// =============================================================================
// 段 2: 三轴伺服电流监测（仅使能时读 AD，%IW×%ID/1e6）
// %IW10/%ID4=俯仰, %IW20/%ID9=方位, %IW30/%ID14=倾斜
// =============================================================================
IF Axis1Status.bServo_Enable THEN
	rELCurrent:=DINT_TO_REAL((INT_TO_DINT(%IW10)* %ID4))/1000000.0;  //俯仰轴电流监测
ELSE
	rELCurrent:=0;
END_IF

IF Axis2Status.bServo_Enable THEN
	rAzCurrent:=DINT_TO_REAL((INT_TO_DINT(%IW20)* %ID9))/1000000.0;  //方位轴电流监测
ELSE
	rAzCurrent:=0;
END_IF

IF Axis3Status.bServo_Enable THEN
	rTlCurrent:=DINT_TO_REAL((INT_TO_DINT(%IW30)* %ID14))/1000000.0;  //倾斜轴电流监测
ELSE
	rTlCurrent:=0;
END_IF

// =============================================================================
// 段 3: 跟踪误差（供 SpiralScan 判断扫描方向与完成度）
// mode2 指向: 命令位置 vs 实际位置
// mode4 程引: 插值目标+偏置 vs 实际位置（含手动/自跟踪偏置）
// =============================================================================
IF Axis2Remote.iMode = 2 THEN
	AzError:=(-1) * (Axis2Remote.rPosCmd-rFctPosReal_2);
	ElError:=Axis1Remote.rPosCmd-rFctPosReal_1;	
END_IF

IF Axis2Remote.iMode = 4 THEN
	AzError:=rFctPosReal_2-RealTimePosCal.rInterazPos-(az_ctrl_1.rStepBias+az_ctrl_1.rAuToStepBias);
	ElError:=RealTimePosCal.rInterElPos-rFctPosReal_1+ (El_ctrl_1.rStepBias+EL_ctrl_1.rAuToStepBias);
END_IF
(*
rAzErrorReal := rAzErrorReal + rAlpha * (AzError - rAzErrorReal);
rElErrorReal := rElErrorReal + rAlpha * (ElError - rElErrorReal);
*)

// =============================================================================
// 段 4: 远控故障复位（Modbus bCommReset → GVL.bError_Reset）
// =============================================================================
IF NOT GVL.bLocalCtrl THEN
	IF Modbus_Slave.bCommReset THEN
		GVL.bError_Reset:=TRUE;
	ELSE
		GVL.bError_Reset:=FALSE;
	END_IF
END_IF

// =============================================================================
// 段 5: 远控 rPosCmd 赋值（含 AGC 搜索偏置或测试扫描偏置）
// 非 bSearch: Modbus 目标 + eltest/aztest
// bSearch:   Modbus 目标 + *_ctrl_1 的 rSearchNextStepTarget_tb
// =============================================================================
IF NOT modbus_slave.bSearch THEN
	Axis1Remote.rPosCmd:=Modbus_Slave.rPosCmd_1 + eltest;
	Axis2Remote.rPosCmd:=Modbus_Slave.rPosCmd_2 - aztest;
ELSE
	Axis1Remote.rPosCmd:=Modbus_Slave.rPosCmd_1 + El_ctrl_1.rSearchNextStepTarget_tb;
	Axis2Remote.rPosCmd:=Modbus_Slave.rPosCmd_2 + Az_ctrl_1.rSearchNextStepTarget_tb;
END_IF

// =============================================================================
// 段 6: 远控三轴命令参量 — Modbus_Slave → AxisXRemote（核心汇总）
// 俯仰/方位 rPosCmd 已在段 5 赋值；此处写 mode/速度/PID/加减速等
// =============================================================================
Axis1Remote.iMode:=Modbus_Slave.iMode_1;
Axis1Remote.rVelCmd:=Modbus_Slave.rVelcmd_1;
//Axis1Remote.rPosCmd:=Modbus_Slave.rPosCmd_1;
Axis1Remote.rP:=Modbus_Slave.rP_1;
Axis1Remote.rI:=Modbus_Slave.rI_1;
Axis1Remote.rD:=Modbus_Slave.rD_1;
Axis1Remote.rPIDThre:=Modbus_Slave.rThreshold_1;
Axis1Remote.rAcceleration:=Modbus_Slave.rAcceleration_1;
Axis1Remote.rDeceleration:=Modbus_Slave.rDeceleration_1;
Axis1Remote.rVel_Limit:=Modbus_Slave.rVelLim_1;

Axis2Remote.iMode:=Modbus_Slave.iMode_2;
Axis2Remote.rVelCmd:=Modbus_Slave.rVelcmd_2;
//Axis2Remote.rPosCmd:=Modbus_Slave.rPosCmd_2;
Axis2Remote.rP:=Modbus_Slave.rP_2;
Axis2Remote.rI:=Modbus_Slave.rI_2;
Axis2Remote.rD:=Modbus_Slave.rD_2;
Axis2Remote.rPIDThre:=Modbus_Slave.rThreshold_2;
Axis2Remote.rAcceleration:=Modbus_Slave.rAcceleration_2;
Axis2Remote.rDeceleration:=Modbus_Slave.rDeceleration_2;
Axis2Remote.rVel_Limit:=Modbus_Slave.rVelLim_2;

Axis3Remote.iMode:=Modbus_Slave.iMode_3;
Axis3Remote.rVelCmd:=Modbus_Slave.rVelcmd_3;
Axis3Remote.rPosCmd:=Modbus_Slave.rPosCmd_3;
Axis3Remote.rP:=Modbus_Slave.rP_3;
Axis3Remote.rI:=Modbus_Slave.rI_3;
Axis3Remote.rD:=Modbus_Slave.rD_3;
Axis3Remote.rPIDThre:=Modbus_Slave.rThreshold_3;
Axis3Remote.rAcceleration:=Modbus_Slave.rAcceleration_3;
Axis3Remote.rDeceleration:=Modbus_Slave.rDeceleration_3;

(* 本控 HMI 赋值块已注释，本控参数由其他 POU 写入 AxisXLocal *)

// =============================================================================
// 段 7: 俯仰预限位 → Error_code 201(正)/202(负)，置位上报标志
// bPrelimit_1 由硬件 IO 映射；触发后根据当前位置方向区分正负限位
// =============================================================================
IF bPrelimit_1 THEN
	IF rFctPosReal_1>0 THEN
		bPrelimit_Positive_1:=TRUE;
		Error_code:=201;
	ELSE
		bPrelimit_Negative_1:=TRUE;
		Error_code:=202;
	END_IF;
ELSE
	bPrelimit_Negative_1:=FALSE;
	bPrelimit_Positive_1:=FALSE;
	;
END_IF

// =============================================================================
// 段 8: 方位预限位（仅置标志，Error_code 203/204 已注释）
// =============================================================================
IF bPrelimit_2 THEN
	IF rFctPosReal_2>0 THEN
		//Error_code:=203;
		bPrelimit_Positive_2:=TRUE;;
	ELSE
		//Error_code:=204;
		bPrelimit_Negative_2:=TRUE;;
	END_IF;
ELSE
	bPrelimit_Negative_2:=FALSE;
	bPrelimit_Positive_2:=FALSE;
	;
END_IF

// =============================================================================
// 段 9: 扫描找到中心 — 基带锁 且 Eb/N0>rEbN0LockThre 且 √(Ua²+Ue²)<=rErrorThre
// =============================================================================
bBaseLock := (READ_485.recBuf[1] = 1);
bErrorLock  := (SQRT(GVL.Chan1Ua * GVL.Chan1Ua + GVL.Chan1Ue * GVL.Chan1Ue) <= PersistentVars.rErrorThre);
bLockSearch := (READ_485.Chan1EB_N0 > PersistentVars.rEbN0LockThre) AND bBaseLock AND bErrorLock;

// =============================================================================
// 段 10: 启扫 — 双轴程引、未自跟踪、基带锁连续 2s（200×10ms）触发一次
// 扫描过程中允许短暂掉锁；找到合格点后本程引周期内不再重扫
// 退出程引则清锁存
// =============================================================================
IF Axis1Remote.iMode = 4 AND Axis2Remote.iMode = 4 THEN
	IF NOT GVL.bStartTrack AND NOT bScanRun AND NOT bScanFound THEN
		IF bBaseLock THEN
			icountBaseLock := icountBaseLock + 1;
			IF icountBaseLock >= 200 THEN
				icountBaseLock := 200;
				bScanRun := TRUE;
			END_IF
		ELSE
			icountBaseLock := 0;
		END_IF
	ELSE
		icountBaseLock := 0;
	END_IF
	enable := bScanRun AND NOT GVL.bStartTrack;
ELSE
	enable := FALSE;
	bScanRun := FALSE;
	bScanDoneOnce := FALSE;
	bScanFound := FALSE;
	az_latch := 0.0;
	el_latch := 0.0;
	icountBaseLock := 0;
END_IF

// 螺旋局部参数（与直线 PersistentVars.rStep 量纲不同：此处为每格周期数）
IF rdelta < 1.0E-6 THEN
	rdelta := 0.25;
END_IF
IF rStep < 1.0E-6 THEN
	rStep := 12.0;
END_IF

// =============================================================================
// 段 11: 调用扫描 FB — 直线或螺旋；locked=找到中心，连续10拍（约100ms）锁存
// =============================================================================
IF NOT PersistentVars.bSearchType THEN
	fbScan(
		enable      := enable,
		delta       := PersistentVars.rAzScanRange,
		delta1      := PersistentVars.rElScanRange,
		n_steps     := PersistentVars.rStep,
		agc      := READ_485.Chan1EB_N0,
		locked     := bLockSearch,
		AzError := AzError,
		elError := elError,
		bTrackState := GVL.bStartTrack,
		azimuth     => az_out,
		elevation   => el_out,
		done        => done_out,
		bType  =>bType_out
	);
ELSE
	fbScan1(
		enable      := enable,
		delta       := rdelta,
		n_steps     := rStep,
		agc      := READ_485.Chan1EB_N0,
		locked     := bLockSearch,
		AzError := AzError,
		elError := elError,
		azimuth     => az_out,
		elevation   => el_out,
		done        => done_out,
		bType  =>bType_out
	);
END_IF

// 扫描结束：找到则锁存 -Error；未找到锁存 0。此后 az_out/el_out 用锁存值
IF bScanRun AND done_out THEN
	bScanRun := FALSE;
	bScanDoneOnce := TRUE;
	IF bType_out THEN
		az_latch := az_out;
		el_latch := el_out;
		bScanFound := TRUE;
	ELSE
		az_latch := 0.0;
		el_latch := 0.0;
		bScanFound := FALSE;
	END_IF
END_IF
IF GVL.bStartTrack AND bScanRun THEN
	bScanRun := FALSE;
	bScanDoneOnce := TRUE;
END_IF
IF NOT bScanRun THEN
	az_out := az_latch;
	el_out := el_latch;
END_IF

// =============================================================================
// 段 12: 自跟踪只跟 ACU HR[7].B10（上升沿开、下降沿关），扫描结束不置位
// =============================================================================
IF Axis1Remote.iMode = 4 AND Axis2Remote.iMode = 4 THEN
	RiseEdge(CLK := Modbus_Slave.bStartTrackAcu);
	FallEdge(CLK := Modbus_Slave.bStartTrackAcu);
	IF RiseEdge.Q THEN
		GVL.bStartTrack := TRUE;
	END_IF;
	IF FallEdge.Q THEN
		GVL.bStartTrack := FALSE;
	END_IF;
ELSE
	GVL.bStartTrack := Modbus_Slave.bStartTrackAcu;
	icountLostLocking := 0;
	icountLostLocking1 := 0;
	Iconutwait := 0;
END_IF

(* fbScantest 测试块已注释 *)

(* PHASE_CAL_HOOK: once per 10 ms, LAST call. *)
PRG_PhaseCalibration();
                  
END_PROGRAM

FUNCTION_BLOCK PID_1
VAR_INPUT
    rTarget : REAL;       (* 设定值 *)
    rFeedback : REAL;       (* 反馈值 *)
	rPosLimPositive:LREAL;//位置正限位
	rPosLimNegative:LREAL;//位置反限位
	rKp:REAL;     //比例增益
	rKi:REAL;     //积分增益
	rKd:REAL;     //微分增益
	iThreshold:INT;//积分项开启的位置阈值
	bPIDEnable:BOOL:=TRUE;//PID使能
	rVelLim:LREAL;//速度限制
END_VAR
VAR_OUTPUT
    rPIDOutput : LREAL:=0;         //带方向的输出速度

END_VAR
VAR
	//rPIDOutPut: REAL:=0.0;
	rLastError: LREAL:=0.0;(*上一次误差*)
	rErrorNow:LREAL:=0.0;(*当前误差*)
    rIntegralNew : LREAL := 0.0; (* 积分项 *)
    rDerivativeNew : LREAL := 0.0; (* 微分项 *)
	rDelta: LREAL;(*增量*)
	rProportionNew: LREAL;
	
	//iAzPIDEnable: INT;
END_VAR

                    
IF (bPIDEnable>0) THEN //如果PID使能
	IF rTarget=rFeedback THEN
		rPIDOutput:=0;	
	ELSE
	
		rErrorNow:=rTarget-rFeedback;//计算当前误差 en
		rProportionNew:=rErrorNow;//比例项
		//积分项
		IF rFeedback>rPosLimNegative AND rFeedback<rPosLimPositive THEN //若在软限位之内，工作时开启积分项
			IF (ABS(rTarget-rFeedback)<iThreshold OR iThreshold = -1) THEN//位置差小于积分阈值开始积分，或者设置阈值为-1，不启用这个控制
				rIntegralNew:= rIntegralNew+rErrorNow; //积分项
			ELSE
				rIntegralNew:=0;
			END_IF;
		ELSE //不在软限位范围内,则积分项为0
			rIntegralNew:=0;
		END_IF

		//PID输出
		rPIDOutPut:=rKp*rProportionNew+rKi*rIntegralNew;


		//PID限速
		
			IF rPIDOutput<(-rVelLim) THEN
				rPIDOutput:=-rVelLim;
			ELSIF rPIDOutput>rVelLim THEN
				rPIDOutput:=rVelLim;
			END_IF
		
		
		IF rFeedback>rPosLimPositive AND rPIDOutput>0 THEN 
			rPIDOutput:=0;
		END_IF
		IF rFeedback<rPosLimNegative AND rPIDOutput<0 THEN
			rPIDOutput:=0;
		END_IF
		
		rLastError:=rErrorNow;//将当前误差赋值给上一次误差
		
	END_IF
ELSE//非使能清零PID各项
	rProportionNew:=0.0;
	rIntegralNew:=0.0;
	rPIDOutput:=0.0;
END_IF










                  
END_FUNCTION_BLOCK

PROGRAM AutoTrackingCal
VAR
	rChanUa:REAL;//自跟踪采用的跟踪接收机ua
	rChanUe:REAL;//自跟踪采用的跟踪接收机ue
	rChanAGC:REAL;//自跟踪采用的跟踪接收机AGC
	bChanLock:BOOL;//频道是否锁定
	iCountATLock:INT;//自跟踪锁定
	iState:INT;//Case选择变量
	
	rAzSum:LREAL;//方位累计量
	rElSum:LREAL;//俯仰累积量
	
	rDirSenFac:REAL:=12;
	rCurentEl:LREAL;//当前俯仰角
	rk: LREAL:=1/15.0;
	
	rChanUaLocal:REAL;//自跟踪采用的跟踪接收机ua
	rChanUeLocal:REAL;//自跟踪采用的跟踪接收机ue
END_VAR

                    (*
IF iState=1 THEN
	rChanUa:=GVL.Chan1Ua;
	rChanUe:=GVL.Chan1Ue;
	rChanAGC:=GVL.Chan1AGC;
	bChanLock:=TRUE;
ELSIF iState=2 THEN
	rChanUa:=GVL.Chan2Ua;
	rChanUe:=GVL.Chan2Ue;
	rChanAGC:=GVL.Chan2AGC;
	bChanLock:=TRUE;
ELSE 
	bChanLock:=FALSE;
END_IF
*)

//iState:=modbusSlave.Trace_Num;//跟踪支路选择
iState:=1;

CASE iState OF 
	1://使用跟踪接收机1 且锁定标识为True
		//
		//bChanLock:=TRUE;
		//方位
		IF GVL.bStartTrack AND (GVL.Chan1Lock OR Securitycheck.bErrorLock) THEN
			//根据误差电压正负决定拉偏方向
			rChanUa:=GVL.Chan1Ua;
			//rChanUa:=rChanUa/UDINT_TO_REAL(modbusSlave.DirSenFac);
			rChanUa:=rChanUa/rDirSenFac;
			rCurentEl:=(rFctPosReal_1-90)*3.1415926535897/180.0;
			rChanUa:=rChanUa/COS(rCurentEl);
			
			//俯仰
			rChanUe:=GVL.Chan1Ue;
			//rChanUe:=rChanUe/UDINT_TO_REAL(modbusSlave.DirSenFac);;
			rChanUe:=rChanUe/rDirSenFac;
			rChanAGC:=GVL.Chan1AGC;
			
			//累积量
			rAzSum:=rAzSum+rk*rChanUa/1000.0;
			rElSum:=rElSum+rk*rChanUe/1000.0;
		ELSE
			rAzSum:=0;
			rElSum:=0;
			rChanUa:=0;
			rChanUe:=0;
		END_IF
		
	2://使用跟踪接收机2 且锁定标识为True
		//
		//bChanLock:=TRUE;
		rChanUa:=GVL.Chan2Ua;
		rChanUe:=GVL.Chan2Ue;
		rChanAGC:=GVL.Chan2AGC;
		//跟踪接收机拉偏量
		(*
		rChanUa:=GVL.Chan2Ua/modbusSlave.DirSenFac;
		rChanUe:=GVL.Chan2Ue/modbusSlave.DirSenFac;
		*)
	3://锁定标识符为False
		//
		//bChanLock:=FALSE;
END_CASE
                  
END_PROGRAM

PROGRAM Ti_ctrl_1
VAR
	Axis3_Ctrl:Ti_Ctrl_FB;
	bRemote2LocalStop:BOOL;
	bLocal2RemoteStop:BOOL;
	Error:INT;
	
	Axis3Limit_pos:REAL;//正软限位
	Axis3Limit_Neg:REAL;//负软限位
	
	bRTriger:Standard.R_TRIG;//本控上升沿
	bFTriger:Standard.F_TRIG;//远控下降沿
	Stop3_Count: INT;
	bStop_3: BOOL;
	
	//指向模式自跟踪
	rPosModeStepBias:LREAL;//指向模式自跟踪拉偏累计值
	rPosModeStep:LREAL:=0.005;//指向模式自跟踪步长，积分用
	rStepBiasMax:LREAL:=2;//指向模式拉偏最大值
	
	//程引拉偏
	rStepBias:LREAL;//步进拉偏累计值
// 	rStep:LREAL:=0.0002;//步长，与控制周期有关，1ms周期对应1秒内累积0.0002*1000=0.2°
// 	rStep:LREAL:=0.01;//步长，与控制周期有关，50ms周期对应1秒内累积0.01*20=0.2°
	rStep:LREAL:=0.004;//步长，与控制周期有关，20ms周期对应1秒内累积0.004*50=0.2°
		
	//自跟踪拉偏
	rAuToStepBias:LREAL;//步进拉偏累计值
// 	rAutoStep:LREAL:=0.005;//步长
	rAutoStep:LREAL:=0.01;//步长
	TbAutoTrigger:Standard.F_TRIG;//自跟踪关闭的下降沿
	RbAutoTrigger:Standard.R_TRIG;//自跟踪开启的上升沿

	rAutoTrackingBiasMax:LREAL:=300;//自跟踪拉偏最大值
	rLocalInitPosModeSpeed: REAL;
	rRemoteInitPosModeSpeed: REAL;
	iCountOffAuto: INT;
	
	iCasePBAutoTrack:INT:=2;//程序引导自跟踪切换 
// 	rKAuToStepBias:LREAL:=0.25;
	rKAuToStepBias:LREAL:=0.16;
	bVisError:BOOL; //报错可视化标识
END_VAR

                    IF GVL.Error_code <> 0 THEN
	bVisError := TRUE;
ELSE
	bVisError := FALSE;
END_IF
(*
//远控轴参量赋值
Axis2Remote.iMode:=Modbus_Slave.iMode_2;
Axis2Remote.rVelCmd:=Modbus_Slave.rVelcmd_2;
Axis2Remote.rPosCmd:=Modbus_Slave.rPosCmd_2;
Axis2Remote.rP:=Modbus_Slave.rP_2;
Axis2Remote.rI:=Modbus_Slave.rI_2;
Axis2Remote.rD:=Modbus_Slave.rD_2;
Axis2Remote.rPIDThre:=Modbus_Slave.rThreshold_2;
Axis2Remote.rAcceleration:=Modbus_Slave.rAcceleration_2;
Axis2Remote.rDeceleration:=Modbus_Slave.rDeceleration_2;
Axis2Remote.rVel_Limit:=Modbus_Slave.rVelLim_2;
*)
// 倾斜轴状态写入
Axis3Status.Error := GVL.bTiStsBit3;
Axis3Status.ErrorID := GVL.eTiErrorcode;
Axis3Status.bServo_Enable := GVL.bTiStsBit0 AND GVL.bTiStsBit1 AND GVL.bTiStsBit2;
Axis3Status.bBrake := NOT (GVL.bTiStsBit0 AND GVL.bTiStsBit1 AND GVL.bTiStsBit2);
Axis3Status.Disabled := NOT (GVL.bTiStsBit0 AND GVL.bTiStsBit1 AND GVL.bTiStsBit2);
Axis3Remote.rSoft_limit_Negative:=-190;Axis3Remote.rSoft_limit_Postive:=190;
Axis3Local.rSoft_limit_Negative:=-190;Axis3Local.rSoft_limit_Postive:=190;

//速度的写入
rFctVelReal_3:=DINT_TO_REAL(diTiActVel)/524288.0*360.0;
//位置的写入，方位0对应编码器0，所以实际方位是：-1*编码器值
//rFctPosReal_3:=DINT_TO_REAL(diTiActPos)/524288.0*360.0-11.413-0.08;
rFctPosReal_3:=DINT_TO_REAL(diTiActPos)/524288.0*360.0;
//软限位控制
Axis3Limit_pos:=190;
Axis3Limit_Neg:=-190;
IF Axis3Remote.rPosCmd>Axis3Limit_pos THEN
	Axis3Remote.rPosCmd:=190;
ELSIF Axis3Remote.rPosCmd<Axis3Limit_Neg THEN
	 Axis3Remote.rPosCmd:=-190;  
END_IF

IF Axis3Local.rPosCmd>Axis3Limit_pos THEN
	Axis2Local.rPosCmd:=190;
ELSIF Axis3Local.rPosCmd<Axis3Limit_Neg THEN
	 Axis3Local.rPosCmd:=-190;  
END_IF

//停止标志符号判断
IF  ABS(rFctVelReal_3)<0.035 THEN
	Stop3_Count:=Stop3_Count+1;
	IF Stop3_Count>100 THEN
		Stop3_Count:=101;
		bStop_3:=TRUE;;
	END_IF
ELSE
	Stop3_Count:=0;
	bStop_3:=FALSE;
END_IF
Axis3Status.Moving := NOT bStop_3;
//PID使能赋值
IF Axis3Remote.iMode=2 OR Axis3Remote.iMode=4 THEN
	Axis3Remote.bPIDEnable:=TRUE;
ELSE
	Axis3Remote.bPIDEnable:=FALSE;
END_IF

//本远控逻辑保护
//远控切本控逻辑保护
bRTriger(CLK:=GVL.bLocalCtrl);
bFTriger(CLK:=GVL.bLocalCtrl);

IF Axis3Status.bServo_Enable AND (bRTriger.Q ) THEN//如果速度不为0且本控发生切换，则减速停止标识为True
	bRemote2LocalStop:=TRUE;
END_IF
IF bRemote2LocalStop  THEN //若减速停止标识符为True 
	
	IF  bStop_3=TRUE THEN//且电机速度不为0 开始减速 减速完成后下使能，下使能完成后复位标识符复位
		Axis3Local.iMode:=0;
		Axis3Remote.iMode:=0;
		IF Axis3Status.bServo_Enable=FALSE THEN
			bRemote2LocalStop:=FALSE;
		END_IF
	ELSE
		Axis3Remote.iMode:=7;
	END_IF
END_IF

//本控切远控
IF Axis3Status.bServo_Enable AND (bFTriger.Q ) THEN//如果速度不为0且本控发生切换，则减速停止标识为True
	bLocal2RemoteStop:=TRUE;
END_IF
IF bLocal2RemoteStop  THEN //若减速停止标识符为True 
	
	IF  bStop_3=TRUE THEN//且电机速度不为0 开始减速 减速完成后下使能，下使能完成后复位标识符复位
		Axis3Local.iMode:=0;
		Axis3Remote.iMode:=0;
		IF Axis3Status.bServo_Enable=FALSE THEN
			bLocal2RemoteStop:=FALSE;
		END_IF
	ELSE
		Axis3Remote.iMode:=7;
		Axis3Local.iMode:=7;
	END_IF
END_IF
(*
//自跟踪
IF GVL.bStartTrack THEN
	Axis2Remote.bStartAutoTrack := TRUE;
	Axis2Remote.rChanU := -AutoTrackingCal.rChanUa;
ELSE
	Axis2Remote.bStartAutoTrack := FALSE;	
	Axis2Remote.rChanU := 0;
END_IF
//拉偏
Axis2Remote.rPIDCmdPos:=RealTimePosCal.rInterAzPos+Modbus_Slave.rBias_2;
*)
//限位
IF Axis3Remote.rPIDCmdPos<-190 THEN
	Axis3Remote.rPIDCmdPos:=-190;
ELSIF Axis3Remote.rPIDCmdPos>190 THEN
	Axis3Remote.rPIDCmdPos:=190;
END_IF

Axis3_Ctrl(sLocal:=Axis3Local, sCtrl:=Axis3Remote, sStatus:=Axis3Status, sVisible:=Axis3Visible, rRealPos:=rFctPosReal_3, rPosLimK:=0.34);
	

                  
END_PROGRAM

FUNCTION_BLOCK Ti_Ctrl_FB
VAR_INPUT
	sLocal:AxisCrtlStruct;
	sCtrl:AxisCrtlStruct;
	sStatus:AxisStatus;
	sVisible:AxisVisible;
	rRealPos:REAL;
	rPosLimK:REAL;
END_VAR
VAR_OUTPUT
	logicError:INT;
END_VAR
VAR
	VelPID_1:PID;
	VelPID_2:PID;
	TON_0:TON;
	bTick:BOOL;
	tr:BOOL;
	icount1:INT := 0;
	icount2:INT := 0;
	icount3:INT := 0;
	bfin1:BOOL;
	bfin2:BOOL;
	istate:INT:=0;
	icount:INT:=0;
END_VAR

                    // 下电时复位控制字bit8
IF sStatus.Disabled OR(NOT sStatus.Moving)THEN
	bTiCtrlBit8 := FALSE;
END_IF

//	错误复位功能
IF GVL.bError_Reset THEN
	sCtrl.iMode:=6;
	sLocal.iMode:=6;
	GVL.Error_code:=0;
END_IF
IF GVL.Error_code =0 THEN
	GVL.bError_Reset:=FALSE;
END_IF

/////////心跳报错清除/////////
IF GVL.eTiErrorcode = 16#8130 AND NOT tr THEN
	GVL.bTiCtrlBit7 := TRUE;
	tr:=TRUE;
	istate:=0;
	icount:=0;
	// 写入下电控制字
	GVL.bTiCtrlBit3 := FALSE;
	GVL.bTiCtrlBit0 := FALSE;
	GVL.bTiCtrlBit1 := FALSE;
	GVL.bTiCtrlBit2 := FALSE;
END_IF
IF tr THEN
	icount1 := icount1 + 1;
END_IF
IF icount1 > 101 THEN
	icount1 := 0;
	tr := FALSE;
	GVL.bTiCtrlBit7 := FALSE;
	bfin1 := TRUE;
END_IF
IF bfin1 THEN
	icount2 := icount2 + 1;
END_IF
IF icount2 > 101 THEN
	bfin1 := FALSE;
	icount2 := 0;
END_IF
/////////////////////////////

IF GVL.Error_code=0 AND GVL.eTiErrorcode = 0 AND NOT GVL.bTiCtrlBit7  AND NOT tr AND NOT bfin1 AND NOT bfin2 THEN
	IF GVL.bLocalCtrl=FALSE THEN //远控
		IF sCtrl.iMode <> 1 THEN
			istate:=0;
			icount:=0;
		END_IF
		CASE sCtrl.iMode OF
			MODES.powerOff: // 下电
				IF NOT sStatus.Disabled THEN
					IF sStatus.Moving THEN // 运动中，先停止运动
						GVL.diTiTargetVel := 0;
						bTiCtrlBit8 := TRUE;
					ELSE
						// 写入下电控制字
						GVL.bTiCtrlBit3 := FALSE;
						GVL.bTiCtrlBit0 := FALSE;
						GVL.bTiCtrlBit1 := FALSE;
						GVL.bTiCtrlBit2 := FALSE;
					END_IF
				END_IF
			MODES.powerOn:  // 上电
				IF sStatus.Disabled THEN
					// 目标速度清零
					GVL.diTiTargetVel := 0;
					IF GVL.siTiMode <> 3 THEN // 上电时模式默认为3，速度模式
						GVL.siTiMode := 3;
					END_IF
					IF siTiMode = 3 THEN
						CASE istate OF
							0:
								GVL.bTiCtrlBit1 := TRUE;
								GVL.bTiCtrlBit2 := TRUE;
								icount := icount + 1;
								IF icount = 20 THEN
									icount:=0;
									istate:=1;
								END_IF
							1:
								GVL.bTiCtrlBit0 := TRUE;
								icount := icount + 1;
								IF icount = 20 THEN
									icount:=0;
									istate:=2;
								END_IF
							2:
								GVL.bTiCtrlBit3 := TRUE;
						END_CASE
					END_IF
				ELSE
					IF sStatus.Moving THEN
						GVL.diTiTargetVel := 0;
						bTiCtrlBit8 := TRUE;
					ELSE
						bTiCtrlBit8 := FALSE;
					END_IF
				END_IF
			MODES.positionMode: // 远控指向模式
				IF NOT sStatus.Disabled THEN
					IF sCtrl.bStartAutoTrack THEN
						(*
						//自跟踪模式下，由误差电压直接驱动
						VelPID_1(rTarget:=sCtrl.rChanU + rRealPos,
								rFeedback:=rRealPos,
								rPosLimPositive:=sCtrl.rSoft_limit_Postive,
								rPosLimNegative:=sCtrl.rSoft_limit_Negative,
								rVelLim:=sCtrl.rVel_Limit,
								rKp:=sCtrl.rP_AutoTrack,//自跟踪PI系数3,0.02
								rKi:=sCtrl.rI_AutoTrack,
								rKd:=sCtrl.rD,
								bPIDEnable:=sCtrl.bPIDEnable,
								iThreshold:= -1,
								rPIDOutput=>sCtrl.rPIDCmdVel);
*)							
					ELSE
						//PID计算速度指令
						VelPID_1(rTarget:=sCtrl.rPosCmd,
							rFeedback:=rRealPos,
							rVelLim:=sCtrl.Pos_Vel,
							rPosLimPositive:=sCtrl.rSoft_limit_Postive,
							rPosLimNegative:=sCtrl.rSoft_limit_Negative,
							rKp:=0.8,//程引PI系数地带：1,0.002  高带：3,0.02
							rKi:=0,
							rKd:=0,
							bPIDEnable:=sCtrl.bPIDEnable,
							iThreshold:=sCtrl.rPIDThre,
							rPIDOutput=>sCtrl.rPIDCmdVel);
					END_IF
					GVL.diTiTargetVel := REAL_TO_DINT(sCtrl.rPIDCmdVel * 524288 / 360);
					GVL.diTiTargetAcc := REAL_TO_UDINT(10 * 524288 / 360);   //加速度
					GVL.diTiTargetDec := REAL_TO_UDINT(10 * 524288 / 360);   //减速度
				END_IF
			MODES.velocityMode://手控速度模式-远控模式
				IF NOT sStatus.Disabled THEN
					IF ABS(sCtrl.rVelCmd) <= sCtrl.rVel_Limit THEN
						GVL.diTiTargetVel := REAL_TO_DINT(sCtrl.rVelCmd * 524288 / 360);
					ELSIF sCtrl.rVelCmd > sCtrl.rVel_Limit THEN
						GVL.diTiTargetVel := REAL_TO_DINT(sCtrl.rVel_Limit * 524288 / 360);
					ELSE
						GVL.diTiTargetVel := REAL_TO_DINT(-sCtrl.rVel_Limit * 524288 / 360);
					END_IF
					GVL.diTiTargetAcc := REAL_TO_UDINT(sCtrl.rAcceleration * 524288 / 360);   //加速度
					GVL.diTiTargetDec := REAL_TO_UDINT(sCtrl.rDeceleration * 524288 / 360);   //减速度
				END_IF
			MODES.programBootMode://PID速度模式-正常模式 程引
				IF NOT sStatus.Disabled THEN
					IF sCtrl.bStartAutoTrack THEN
						//自跟踪模式下，由误差电压直接驱动
						VelPID_1(rTarget:=sCtrl.rChanU + rRealPos,
								rFeedback:=rRealPos,
								rPosLimPositive:=sCtrl.rSoft_limit_Postive,
								rPosLimNegative:=sCtrl.rSoft_limit_Negative,
								rVelLim:=sCtrl.rVel_Limit,
								rKp:=sCtrl.rP_AutoTrack,//自跟踪PI系数3,0.02
								rKi:=sCtrl.rI_AutoTrack,
								rKd:=sCtrl.rD,
								bPIDEnable:=sCtrl.bPIDEnable,
								iThreshold:= -1,
								rPIDOutput=>sCtrl.rPIDCmdVel);							
					ELSE
						//PID计算速度指令
						VelPID_1(rTarget:=sCtrl.rPIDCmdPos,
							rFeedback:=rRealPos,
							rVelLim:=sCtrl.rVel_Limit,
							rPosLimPositive:=sCtrl.rSoft_limit_Postive,
							rPosLimNegative:=sCtrl.rSoft_limit_Negative,
							rKp:=sCtrl.rP,//程引PI系数地带：1,0.002  高带：3,0.02
							rKi:=sCtrl.rI,
							rKd:=sCtrl.rD,
							bPIDEnable:=sCtrl.bPIDEnable,
							iThreshold:=sCtrl.rPIDThre,
							rPIDOutput=>sCtrl.rPIDCmdVel);
					END_IF
					GVL.diTiTargetVel := REAL_TO_DINT(sCtrl.rPIDCmdVel * 524288 / 360);
					GVL.diTiTargetAcc := REAL_TO_UDINT(sCtrl.rAcceleration * 524288 / 360);   //加速度
					GVL.diTiTargetDec := REAL_TO_UDINT(sCtrl.rDeceleration * 524288 / 360);   //减速度
				END_IF
			MODES.reset://重置
				IF NOT sStatus.Disabled THEN
					IF sStatus.Moving THEN
						GVL.diTiTargetVel := 0;
						bTiCtrlBit8 := TRUE;
					ELSE
						bTiCtrlBit8 := FALSE;
					END_IF
				END_IF
			MODES.halt://待机
				IF NOT sStatus.Disabled THEN
					IF sStatus.Moving THEN
						GVL.diTiTargetVel := 0;
						bTiCtrlBit8 := TRUE;
					ELSE
						bTiCtrlBit8 := FALSE;
					END_IF
				END_IF
			
		END_CASE
	ELSE // 本控
		IF sLocal.iMode <> 1 THEN
			istate:=0;
			icount:=0;
		END_IF
		CASE sLocal.iMode OF
			MODES.powerOff: // 下电
				IF NOT sStatus.Disabled THEN
					IF sStatus.Moving THEN // 运动中，先停止运动
						GVL.diTiTargetVel := 0;
						bTiCtrlBit8 := TRUE;
					ELSE
						// 写入下电控制字
						GVL.bTiCtrlBit3 := FALSE;
						GVL.bTiCtrlBit0 := FALSE;
						GVL.bTiCtrlBit1 := FALSE;
						GVL.bTiCtrlBit2 := FALSE;
					END_IF
				END_IF
			MODES.powerOn:  // 上电
				IF sStatus.Disabled THEN
					// 目标速度清零
					GVL.diTiTargetVel := 0;
					IF GVL.siTiMode <> 3 THEN // 上电时模式默认为3，速度模式
						GVL.siTiMode := 3;
					END_IF
					IF siTiMode = 3 THEN
						CASE istate OF
							0:
								GVL.bTiCtrlBit1 := TRUE;
								GVL.bTiCtrlBit2 := TRUE;
								icount := icount + 1;
								IF icount = 20 THEN
									icount:=0;
									istate:=1;
								END_IF
							1:
								GVL.bTiCtrlBit0 := TRUE;
								icount := icount + 1;
								IF icount = 20 THEN
									icount:=0;
									istate:=2;
								END_IF
							2:
								GVL.bTiCtrlBit3 := TRUE;
						END_CASE
					END_IF
				ELSE
					IF sStatus.Moving THEN
						GVL.diTiTargetVel := 0;
						bTiCtrlBit8 := TRUE;
					ELSE
						bTiCtrlBit8 := FALSE;
					END_IF
				END_IF
			MODES.velocityMode://手控速度模式-本控模式
				IF NOT sStatus.Disabled THEN
					IF ABS(sLocal.rVelCmd) <= sLocal.rVel_Limit THEN
						GVL.diTiTargetVel := REAL_TO_DINT(sLocal.rVelCmd * 524288 / 360);
					ELSIF sLocal.rVelCmd > sLocal.rVel_Limit THEN
						GVL.diTiTargetVel := REAL_TO_DINT(sLocal.rVel_Limit * 524288 / 360);
					ELSE
						GVL.diTiTargetVel := REAL_TO_DINT(-sLocal.rVel_Limit * 524288 / 360);
					END_IF
					GVL.diTiTargetAcc := REAL_TO_UDINT(sLocal.rAcceleration * 524288 / 360);   //加速度
					GVL.diTiTargetDec := REAL_TO_UDINT(sLocal.rDeceleration * 524288 / 360);   //减速度
				END_IF
			MODES.programBootMode://本控位置模式
				IF NOT sStatus.Disabled THEN
					IF NOT sLocal.bPIDEnable THEN
						GVL.diTiTargetVel := 0;							
					ELSE
						//PID计算速度指令
						 VelPID_2(rTarget:=sLocal.rPosCmd,
							     rFeedback:=rRealPos,
								 rPosLimPositive:=sLocal.rSoft_limit_Postive,//软限位
								 rPosLimNegative:=sLocal.rSoft_limit_Negative,
								 rKp:=sLocal.rP,
								 rKi:=sLocal.rI,
								 rKd:=sLocal.rD,
								 iThreshold:=sLocal.rPIDThre,
								 bPIDEnable:=sLocal.bPIDEnable,
								 rVelLim:=sLocal.Pos_Vel,
								 rPIDOutput=>sLocal.rPIDCmdVel);//普通PID
					END_IF
					GVL.diTiTargetVel := REAL_TO_DINT(sLocal.rPIDCmdVel * 524288 / 360);
					GVL.diTiTargetAcc := REAL_TO_UDINT(sLocal.rAcceleration * 524288 / 360);   //加速度
					GVL.diTiTargetDec := REAL_TO_UDINT(sLocal.rDeceleration * 524288 / 360);   //减速度
				END_IF
			MODES.reset://重置
			// 是否需要
			MODES.halt://待机
				IF NOT sStatus.Disabled THEN
					IF sStatus.Moving THEN
						GVL.diTiTargetVel := 0;
						bTiCtrlBit8 := TRUE;
					ELSE
						bTiCtrlBit8 := FALSE;
					END_IF
				END_IF
			
		END_CASE
	END_IF
ELSIF GVL.Error_code<>0 AND GVL.eTiErrorcode = 0 AND NOT GVL.bTiCtrlBit7  AND NOT tr AND NOT bfin1 AND NOT bfin2 THEN
	// 出现错误，轴停止运动
	GVL.diTiTargetVel := 0;
	bTiCtrlBit8 := TRUE;
	TON_0(IN:=bTiCtrlBit8,PT:=T#1S,Q=>,ET=>);//判断stop0执行是否超时,若超时强制下电（手动复位）
	IF TON_0.Q THEN
		bTick:=TRUE;
	END_IF
	IF bTick AND sStatus.Moving THEN // 超时强制下电
		// 写入下电控制字
		GVL.bTiCtrlBit3 := FALSE;
		GVL.bTiCtrlBit0 := FALSE;
		GVL.bTiCtrlBit1 := FALSE;
		GVL.bTiCtrlBit2 := FALSE;
	END_IF
END_IF
                  
END_FUNCTION_BLOCK

FUNCTION_BLOCK vpid
VAR_INPUT
	rTarget : REAL;           // 设定值
    rFeedback : REAL;         // 反馈值
    rPosLimPositive : LREAL;  // 位置正限位
    rPosLimNegitive : LREAL;  // 位置反限位
    rKpBase : REAL;           // 基础比例增益
    rKiBase : REAL;           // 基础积分增益
    rVelThreshold : LREAL;     // 速度阈值，真实值除以控制频率
    rKpScale : REAL;          // 比例增益比例因子
    rKiScale : REAL;          // 积分增益比例因子
    iThrehold : INT;          // 积分项开启的位置阈值
    bPIDEnable : BOOL := TRUE;// PID使能
    rVelLim : LREAL;          // 速度限制
	rKpMax : REAL;
	rKiMax : REAL;
	rElPos : REAL;            // 俯仰角度
END_VAR

VAR_OUTPUT
    rPIDOutput : LREAL := 0;  // 控制量
	rPIDOutDir: LREAL;
END_VAR

VAR
    rLastFeedback : LREAL := 0.0; // 上一次反馈值
    rErrorNow : LREAL := 0.0;     // 当前误差
    rIntegralNew : LREAL := 0.0;  // 积分项
    rDelta : LREAL;               // 增量
    rProportionNew : LREAL;       // 比例项
    rSpeed : REAL;                // 当前速度
    rKp : REAL:=1;                   // 动态比例增益
    rKi : REAL:=0.02;                   // 动态积分增益
	rInterValueNow : LREAL := 0.0;        // 当前插值位置
	rInterValueLast : LREAL := 0.0;       // 上一次插值位置
	//rSlope :LREAL :=0; 			  //PI变化斜率
	rStep:LREAL:=0.002;                //PI变化率
	
	rKpTarget :REAL:=1;
	rKiTarget :REAL:=0.02;
	
	
END_VAR

                    IF (bPIDEnable) THEN // 如果PID使能
    IF rTarget = rFeedback THEN
        rPIDOutDir := 0;    
    ELSE
        rErrorNow := rTarget - rFeedback; // 计算当前误差
        rProportionNew := rErrorNow;      // 比例项
		
		IF rElPos > rVelThreshold THEN
			rKpTarget := rKpBase + rKpScale * (rElPos - rVelThreshold);
			rKiTarget := rKiBase + rKiScale * (rElPos - rVelThreshold);
		ELSE
			rKpTarget := rKpBase;
			rKiTarget := rKiBase;
		END_IF
//         rInterValueLast := rInterValueNow; // 将当前插值位置值赋值给上一次
// 		rInterValueNow := RealTimePosCal.ElCubicInter.sout*10000.0;
//         // 计算当前速度
//         // rSpeed := ABS(rFeedback - rLastFeedback);
//         rSpeed := ABS(rInterValueNow - rInterValueLast)/10000.0;
// 		
//         // 根据速度调整PI增益
//         IF rSpeed > rVelThreshold THEN
//             rKpTarget := rKpBase + rKpScale * (rSpeed - rVelThreshold);
//             rKiTarget := rKiBase + rKiScale * (rSpeed - rVelThreshold);
//         ELSE
//             rKpTarget := rKpBase;
//             rKiTarget := rKiBase;
//         END_IF
        IF rKpTarget > rKpMax THEN
			rKpTarget := rKpMax;
		END_IF
		IF rKiTarget > rKiMax THEN
			rKiTarget := rKiMax;
		END_IF
		
		IF rKp<=rKpTarget THEN
			rKp:=rKp+rStep;
		ELSE
			rKp:=rKp-rStep;
		END_IF
		IF rKi<=rKiTarget THEN
			rKi:=rKi+(rKiScale/rKpScale)*rStep;
		ELSE
			rKi:=rKi-(rKiScale/rKpScale)*rStep;
		END_IF
	END_IF
        // 积分项
        IF rFeedback > rPosLimNegitive AND rFeedback < rPosLimPositive THEN // 若在软限位之内，工作时开启积分项
            IF (ABS(rTarget - rFeedback) < iThrehold) THEN // 位置差小于积分阈值
                rIntegralNew := rIntegralNew + rErrorNow;  // 积分项
            ELSE
                rIntegralNew := rIntegralNew;  // 积分项
            END_IF;
        ELSE // 不在软限位范围内，则积分项为0
            rIntegralNew := 0;
        END_IF
        (*
        // 防止目标位置与当前位置偏差过大，导致比例项输出太大，引起震动
        IF rKp * rProportionNew > 2 THEN
            rPIDOutput := 2;
        ELSIF rKp * rProportionNew < -2 THEN
            rPIDOutput := -2;
        ELSE
            rPIDOutput := rKp * rProportionNew + rKi * rIntegralNew / 1000.0; // 由于需求积分项过小，因此积分系数在接口数据上除1000
        END_IF
        *)
		rPIDOutput := rKp * rProportionNew + rKi * rIntegralNew; // 由于需求积分项过小，因此积分系数在接口数据上除1000
        // 根据方向设置输出
        IF rPIDOutput < 0 THEN

            rPIDOutDir := rPIDOutput;
        ELSE

            rPIDOutDir := rPIDOutput;
        END_IF
        
        // PID限速
        IF (ABS(rPIDOutDir) > rVelLim) THEN
            IF rPIDOutDir < (-rVelLim) THEN
                rPIDOutDir := -rVelLim;
            ELSIF rPIDOutDir > rVelLim THEN
                rPIDOutDir := rVelLim;
            END_IF
        END_IF
        
        // 位置限位检查
        IF rFeedback > rPosLimPositive AND rPIDOutDir > 0  THEN
            rPIDOutDir := 0;
        END_IF
        IF rFeedback < rPosLimNegitive AND rPIDOutDir <= 0 THEN
            rPIDOutDir := 0;
        END_IF
        
        //rLastFeedback := rFeedback; // 将当前反馈值赋值给上一次反馈值
		//rInterValueLast := rInterValueNow; // 将当前插值位置值赋值给上一次

ELSE // 非使能清零PID各项
    rProportionNew := 0.0;
    rIntegralNew := 0.0;
    rPIDOutDir := 0.0;
    rPIDOutput := 0.0;
END_IF

                  
END_FUNCTION_BLOCK

PROGRAM READ_485
VAR
	com_init:gcan.FB_Com_Init;      		//gcan.FB_Com_Init为串口初始化功能块，可设定串口端口号，串口波特率等参数
	com_read:gcan.FB_Com_Read ;				//gcan.FB_Com_Read为串口接收功能块，用于通过接收串口发送给PLC的数据
	com_write:gcan.FB_Com_Write ;			//gcan.FB_Com_Write为串口发送功能块，用于发送串口数据
	m_uiError:UINT;							//用于承接功能块中报错引脚错误信息的变量
	m_out:BOOL;								//用于承接功能块中完成标志引脚数据的变量
	isFirst:BOOL:=TRUE;						//用于判断初始化只执行一次的逻辑
	mPort:BYTE;								//程序中用作设定串口端口号
	recSize:UINT;							//接收数据长度，单位：字节
	recBuf:ARRAY[0..19] OF BYTE;			//用于存放接收到的串口数据的数组
	recData:ARRAY[0..8] OF BYTE;			//用于存放整帧数据
	wAGC:WORD; // agc，电平值
	iUa:INT; // 方位误差电压，mV
	iUe:INT; // 俯仰误差电压，mV
	iChan1DataLen: UINT;
	chan1_i: INT;
	chan1_j: INT;
	Word2Bit1:Word2Bit;
	Word2Bit2:Word2Bit;
	Word2Bit3:Word2Bit;
	rUagcTemp:REAL;
	rUaTemp:REAL;
	rUeTemp:REAL;
	btest:BOOL;
	btest2:BOOL;
	
	rSData:REAL;
	rQData:REAL;
	Dword2Bit1:Dword2Bit;
	Dword2Bit2:Dword2Bit;
	Chan1EB_N0: REAL;
	bEBN0Lock:BOOL;
	icount0:INT;
END_VAR

                    mPort:=2;								//串口端口号设定，GCAN-PLC-400、GCAN-PLC-510、GCAN-PLC-511，1为232，2为485
										//GCAN-PLC-324、GCAN-PLC-326，1为第一路485，2为第2路485
IF isFirst THEN
	com_init(							//串口初始化功能块
	EN_IN:=TRUE,						//串口初始化功能块使能
	xEnable:=TRUE,						//串口功能使能
	bPort:=mPort,						//串口端口号设定
	uiBaudrate:=19200,					//串口波特率设定
	bParity:=0,							//串口奇偶校验设定，0为无校验，1为奇校验，2为偶检验
	bDatabits:=8,						//数据位设定
	bStopbits:=1,						//停止位设定
	EN_OUT=>m_out,						//串口初始化功能块执行完成标志位
	uiError=>m_uiError);				//串口初始化功能块执行错误信息
	isfirst:=FALSE;						//执行一次初始化后关闭IF的条件使其之后进入ELSE程序段运行

ELSE
	com_read(						//串口读取功能块
	EN_in:=TRUE,					//读取功能块使能，为TRUE执行读取
	bPort:=mPort,					//串口端口号设定
	p_brxdata:=ADR(recBuf),			//读取到的串口数据引脚为指针类型，使用ADR()指向自建数组将数据存放到数组中
	uiMaxsize:=20,					//设定最大读取长度
	EN_out=>m_out,					//串口读取功能块执行完成标志位******功能块执行完成不代表接收完成********
	uiRecSize=>recSize,				//串口接收数据长度，单位：字节，大于0时说明接收到数据可用于判断是否接收
	uierror=>m_uierror);			//串口读取功能块执行错误信息
	
	//GVL.Chan1Lock := BYTE_TO_BOOL(recBuf[1]);
	IF recBuf[1] = 1 AND GVL.Chan1AGC >= GVL.Chanthreshold THEN
		GVL.Chan1Lock := TRUE;
	ELSE
		GVL.Chan1Lock := FALSE;
	END_IF
	Word2Bit1.Apart_Byte[1] := recBuf[2];
	Word2Bit1.Apart_Byte[2] := recBuf[3];
	wAGC:=Word2Bit1.Apart_Word;
	
	Word2Bit2.Apart_Byte[1] := recBuf[4];
	Word2Bit2.Apart_Byte[2] := recBuf[5];
	iUa:=Word2Bit2.Apart_INT;
	
	Word2Bit3.Apart_Byte[1] := recBuf[6];
	Word2Bit3.Apart_Byte[2] := recBuf[7];
	iUe:=Word2Bit3.Apart_INT;
	IF ABS(INT_TO_REAL(iUa) * 5 / 2048) <= 5 AND ABS(INT_TO_REAL(iUe) * 5 / 2048) <= 5 AND ABS((WORD_TO_REAL(wAGC) * 5 / 76)) <=5 THEN
		GVL.Chan1Ua := INT_TO_REAL(iUa) * 5 / 2048;
		GVL.Chan1Ue := INT_TO_REAL(iUe) * 5 / 2048;
		GVL.Chan1AGC := 5 - (WORD_TO_REAL(wAGC) * 5 / 76);
	END_IF
	
	(*
	Dword2Bit1.Apart_Byte[4] := recBuf[8];
	Dword2Bit1.Apart_Byte[3] := recBuf[9];
	Dword2Bit1.Apart_Byte[2] := recBuf[10];
	Dword2Bit1.Apart_Byte[1] := recBuf[11];	
	
	
	Dword2Bit2.Apart_Byte[4] := recBuf[12];
	Dword2Bit2.Apart_Byte[3] := recBuf[13];
	Dword2Bit2.Apart_Byte[2] := recBuf[14];
	Dword2Bit2.Apart_Byte[1] := recBuf[15];	
	*)
	
	Dword2Bit1.Apart_Byte[3] := recBuf[8];
	Dword2Bit1.Apart_Byte[4] := recBuf[9];
	Dword2Bit1.Apart_Byte[1] := recBuf[10];
	Dword2Bit1.Apart_Byte[2] := recBuf[11];	
	
	
	Dword2Bit2.Apart_Byte[3] := recBuf[12];
	Dword2Bit2.Apart_Byte[4] := recBuf[13];
	Dword2Bit2.Apart_Byte[1] := recBuf[14];
	Dword2Bit2.Apart_Byte[2] := recBuf[15];	
	
	rQData:=DWORD_TO_REAL(Dword2Bit2.Apart_DWORD);
	rSData:=DWORD_TO_REAL(Dword2Bit1.Apart_DWORD)-rQData;
	//rSData:=INT_TO_REAL(Dword2Bit1.Apart_INT) - rQData;
	
	IF rSData<>0  AND rQData<>0  THEN
		Chan1EB_N0 := 10*LOG(ABS(rSData/rQData))+3.8;
	ELSE
		Chan1EB_N0 := 0;
	END_IF
	
	//程引、位置模式下，信噪比大于29；或上位机下发自跟踪
	IF ((GVL.Axis1Remote.iMode = 2 OR GVL.Axis1Remote.iMode = 4) AND Chan1EB_N0 >= 29)AND READ_485.recBuf[1] = 1 OR Modbus_Slave.bStartTrackAcu THEN
		icount0:=0;
		bEBN0Lock := TRUE;
	END_IF
	IF ( GVL.Axis1Remote.iMode = 4 or GVL.Axis1Remote.iMode =2 ) AND recBuf[1] = 0 THEN
		icount0:=icount0+1;
	END_IF
	IF icount0 > 400 OR (GVL.Axis1Remote.iMode = 0 OR GVL.Axis1Remote.iMode = 0) THEN
		icount0 := 401;
		bEBN0Lock := FALSE;
	END_IF
(* PHASE_CAL_RX_BEGIN: passive diagnostics; original decoder above is unchanged.
   Assumes each eligible read starts at original recBuf[0]. Not a frame parser.
   Admission requires separate operator protocol/alignment confirmation. *)
GVL_PhaseCal.uiReadSize:=recSize;
GVL_PhaseCal.uiSerialError:=m_uiError;
IF recSize>0 THEN
    IF GVL_PhaseCal.udiReadCount>=4294967294 THEN
        GVL_PhaseCal.udiReadCount:=0;
    END_IF;
    GVL_PhaseCal.udiReadCount:=GVL_PhaseCal.udiReadCount+1;
    IF recSize<16 THEN
        IF GVL_PhaseCal.udiShortReadCount>=4294967294 THEN
            GVL_PhaseCal.udiShortReadCount:=0;
        END_IF;
        GVL_PhaseCal.udiShortReadCount:=GVL_PhaseCal.udiShortReadCount+1;
    END_IF;
END_IF;
IF recSize>=16 AND recSize<=20 AND m_uiError=0 AND
   ABS(INT_TO_REAL(iUa)*5/2048)<=5 AND
   ABS(INT_TO_REAL(iUe)*5/2048)<=5 AND
   ABS(WORD_TO_REAL(wAGC)*5/76)<=5 THEN
    IF GVL_PhaseCal.udiRxSeq>=4294967294 THEN
        GVL_PhaseCal.udiRxSeq:=1;
    ELSE
        GVL_PhaseCal.udiRxSeq:=GVL_PhaseCal.udiRxSeq+1;
    END_IF;
    GVL_PhaseCal.lrRxUa:=REAL_TO_LREAL(GVL.Chan1Ua);
    GVL_PhaseCal.lrRxUe:=REAL_TO_LREAL(GVL.Chan1Ue);
    GVL_PhaseCal.lrRxEbN0:=REAL_TO_LREAL(Chan1EB_N0);
    GVL_PhaseCal.lrRxAz:=-REAL_TO_LREAL(GVL.rFctPosReal_2);
    GVL_PhaseCal.lrRxEl:=REAL_TO_LREAL(GVL.rFctPosReal_1)-90;
    GVL_PhaseCal.xRxLock:=(recBuf[1]=1);
    GVL_PhaseCal.udiRxSeq:=GVL_PhaseCal.udiRxSeq+1;
END_IF;
(* PHASE_CAL_RX_END *)
END_IF
(*
//加校验
iChan1DataLen:=recSize-1; //数据长度
	IF iChan1DataLen > 0 THEN
		FOR chan1_i:=0 TO iChan1DataLen BY 1 DO
			
			IF recBuf[chan1_i] = 16#7E THEN
				chan1_j:=0;
			END_IF
			recData[chan1_j]:=recBuf[chan1_i];
			
			chan1_j:=chan1_j+1;
			IF chan1_j=8 THEN
				Word2Bit1.Apart_Byte[1] := recData[2];
				Word2Bit1.Apart_Byte[2] := recData[3];
				wAGC:=Word2Bit1.Apart_Word;
				
				Word2Bit2.Apart_Byte[1] := recData[4];
				Word2Bit2.Apart_Byte[2] := recData[5];
				iUa:=Word2Bit2.Apart_INT;
				
				Word2Bit3.Apart_Byte[1] := recData[6];
				Word2Bit3.Apart_Byte[2] := recData[7];
				iUe:=Word2Bit3.Apart_INT;
				rUaTemp := INT_TO_REAL(iUa) * 5 / 2048;
				rUeTemp := INT_TO_REAL(iUe) * 5 / 2048;
				rUagcTemp := WORD_TO_REAL(wAGC) * 5 / 76;
				
				IF ABS(rUagcTemp)<=5 AND ABS(rUaTemp)<=5 AND ABS(rUeTemp)<=5THEN 
					GVL.Chan1Ua := rUaTemp;
					GVL.Chan1Ue := rUeTemp;
					GVL.Chan1AGC := rUagcTemp;
					IF recData[1] = 1 THEN
						GVL.Chan1Lock := TRUE;
					ELSE
						GVL.Chan1Lock := FALSE;
					END_IF
				END_IF
(* 
				IF ABS(GVL.Chan1AGC)>5 THEN GVL.Chan1AGC:=5;
				END_IF
				IF ABS(GVL.Chan1Ua)>5 THEN GVL.Chan1Ua:=0;
				END_IF
				IF ABS(GVL.Chan1Ue)>5 THEN GVL.Chan1Ue:=0;
				END_IF
				*)
				chan1_j:=0;
			END_IF
		END_FOR
	END_IF
	
	
END_IF
*)
                  
END_PROGRAM

FUNCTION_BLOCK Get_AZ
VAR_INPUT
	uliRealTime : LREAL; // 当前时间戳，单位毫秒
	lrStartTime : LREAL; // 任务起始时间，单位秒
	rNodeTime1 : REAL;
	rNodeTime2 : REAL;
	rNodeTime3 : REAL;
    rNodeTime4 : REAL;
    rNodeTime5 : REAL;
	rEndTime : REAL;
	lrFun1 : ARRAY[0..10] OF LREAL;
	lrFun2 : ARRAY[0..10] OF LREAL;
	lrFun3 : ARRAY[0..10] OF LREAL;
	lrFun4 : ARRAY[0..10] OF LREAL;
	lrFun5 : ARRAY[0..10] OF LREAL;
	lrFun6 : ARRAY[0..10] OF LREAL;
END_VAR
VAR_OUTPUT
	lrFitResult : LREAL;
END_VAR
VAR
	rDelTime : REAL;
	rRealTime : LREAL;
END_VAR

                    rRealTime := uliRealTime / 1000.0 - lrStartTime/1000.0;


IF rRealTime <= 0.0 THEN
	rDelTime := 0.0;
	lrFitResult := lrFun1[10];
ELSIF rRealTime <= rNodeTime1 THEN
    rDelTime := rRealTime - 0.0;
	lrFitResult := lrFun1[0] * EXPT(rDelTime,10) + lrFun1[1] * EXPT(rDelTime,9) + lrFun1[2] * EXPT(rDelTime,8) + lrFun1[3] * EXPT(rDelTime,7) + lrFun1[4] * EXPT(rDelTime,6) + lrFun1[5] * EXPT(rDelTime,5)
    + lrFun1[6] * EXPT(rDelTime,4) + lrFun1[7] * EXPT(rDelTime,3) + lrFun1[8] * EXPT(rDelTime,2) + lrFun1[9] * rDelTime + lrFun1[10];
ELSIF rRealTime <= rNodeTime2 THEN
    rDelTime := rRealTime - rNodeTime1;
    lrFitResult := lrFun2[0] * EXPT(rDelTime,10) + lrFun2[1] * EXPT(rDelTime,9) + lrFun2[2] * EXPT(rDelTime,8) + lrFun2[3] * EXPT(rDelTime,7) + lrFun2[4] * EXPT(rDelTime,6) + lrFun2[5] * EXPT(rDelTime,5)
    + lrFun2[6] * EXPT(rDelTime,4) + lrFun2[7] * EXPT(rDelTime,3) + lrFun2[8] * EXPT(rDelTime,2) + lrFun2[9] * rDelTime + lrFun2[10];
ELSIF rRealTime <= rNodeTime3 THEN
    rDelTime := rRealTime - rNodeTime2;
    lrFitResult := lrFun3[0] * EXPT(rDelTime,10) + lrFun3[1] * EXPT(rDelTime,9) + lrFun3[2] * EXPT(rDelTime,8) + lrFun3[3] * EXPT(rDelTime,7) + lrFun3[4] * EXPT(rDelTime,6) + lrFun3[5] * EXPT(rDelTime,5)
    + lrFun3[6] * EXPT(rDelTime,4) + lrFun3[7] * EXPT(rDelTime,3) + lrFun3[8] * EXPT(rDelTime,2) + lrFun3[9] * rDelTime + lrFun3[10];
ELSIF rRealTime <= rNodeTime4 THEN
    rDelTime := rRealTime - rNodeTime3;
    lrFitResult := lrFun4[0] * EXPT(rDelTime,10) + lrFun4[1] * EXPT(rDelTime,9) + lrFun4[2] * EXPT(rDelTime,8) + lrFun4[3] * EXPT(rDelTime,7) + lrFun4[4] * EXPT(rDelTime,6) + lrFun4[5] * EXPT(rDelTime,5)
    + lrFun4[6] * EXPT(rDelTime,4) + lrFun4[7] * EXPT(rDelTime,3) + lrFun4[8] * EXPT(rDelTime,2) + lrFun4[9] * rDelTime + lrFun4[10];
ELSIF rRealTime <= rNodeTime5 THEN
    rDelTime := rRealTime - rNodeTime4;
    lrFitResult := lrFun5[0] * EXPT(rDelTime,10) + lrFun5[1] * EXPT(rDelTime,9) + lrFun5[2] * EXPT(rDelTime,8) + lrFun5[3] * EXPT(rDelTime,7) + lrFun5[4] * EXPT(rDelTime,6) + lrFun5[5] * EXPT(rDelTime,5)
    + lrFun5[6] * EXPT(rDelTime,4) + lrFun5[7] * EXPT(rDelTime,3) + lrFun5[8] * EXPT(rDelTime,2) + lrFun5[9] * rDelTime + lrFun5[10];
ELSIF rRealTime <= rEndTime THEN
    rDelTime := rRealTime - rNodeTime5;
    lrFitResult := lrFun6[0] * EXPT(rDelTime,10) + lrFun6[1] * EXPT(rDelTime,9) + lrFun6[2] * EXPT(rDelTime,8) + lrFun6[3] * EXPT(rDelTime,7) + lrFun6[4] * EXPT(rDelTime,6) + lrFun6[5] * EXPT(rDelTime,5)
    + lrFun6[6] * EXPT(rDelTime,4) + lrFun6[7] * EXPT(rDelTime,3) + lrFun6[8] * EXPT(rDelTime,2) + lrFun6[9] * rDelTime + lrFun6[10];
ELSE
    rDelTime := rEndTime - rNodeTime5;
    lrFitResult := lrFun6[0] * EXPT(rDelTime,10) + lrFun6[1] * EXPT(rDelTime,9) + lrFun6[2] * EXPT(rDelTime,8) + lrFun6[3] * EXPT(rDelTime,7) + lrFun6[4] * EXPT(rDelTime,6) + lrFun6[5] * EXPT(rDelTime,5)
    + lrFun6[6] * EXPT(rDelTime,4) + lrFun6[7] * EXPT(rDelTime,3) + lrFun6[8] * EXPT(rDelTime,2) + lrFun6[9] * rDelTime + lrFun6[10];
END_IF

IF lrFitResult>270 THEN
	lrFitResult:=270;
ELSIF lrFitResult<-270 THEN
	lrFitResult:=-270;
END_IF
                  
END_FUNCTION_BLOCK

FUNCTION_BLOCK Get_AZ_1
VAR_INPUT
	uliRealTime : LREAL; // 当前时间戳，单位毫秒
	lrStartTime : LREAL; // 任务起始时间，单位秒
	rNodeTime1 : REAL;
	rNodeTime2 : REAL;
	rNodeTime3 : REAL;
    rNodeTime4 : REAL;
    rNodeTime5 : REAL;
	rEndTime : REAL;
	lrFun1 : ARRAY[0..10] OF LREAL;
	lrFun2 : ARRAY[0..10] OF LREAL;
	lrFun3 : ARRAY[0..10] OF LREAL;
	lrFun4 : ARRAY[0..10] OF LREAL;
	lrFun5 : ARRAY[0..10] OF LREAL;
	lrFun6 : ARRAY[0..10] OF LREAL;
END_VAR
VAR_OUTPUT
	lrFitResult : LREAL;
END_VAR
VAR
	rDelTime : REAL;
	rRealTime : LREAL;
END_VAR

                    rRealTime := uliRealTime / 1000.0 - lrStartTime/1000.0;


IF rRealTime <= 0.0 THEN
	rDelTime := 0.0;
	lrFitResult := lrFun1[10];
ELSIF rRealTime <= rNodeTime1 THEN
    rDelTime := rRealTime - 0.0;
	lrFitResult := lrFun1[0] * EXPT(rDelTime,10) + lrFun1[1] * EXPT(rDelTime,9) + lrFun1[2] * EXPT(rDelTime,8) + lrFun1[3] * EXPT(rDelTime,7) + lrFun1[4] * EXPT(rDelTime,6) + lrFun1[5] * EXPT(rDelTime,5)
    + lrFun1[6] * EXPT(rDelTime,4) + lrFun1[7] * EXPT(rDelTime,3) + lrFun1[8] * EXPT(rDelTime,2) + lrFun1[9] * rDelTime + lrFun1[10];
ELSIF rRealTime <= rNodeTime2 THEN
    rDelTime := rRealTime - rNodeTime1;
    lrFitResult := lrFun2[0] * EXPT(rDelTime,10) + lrFun2[1] * EXPT(rDelTime,9) + lrFun2[2] * EXPT(rDelTime,8) + lrFun2[3] * EXPT(rDelTime,7) + lrFun2[4] * EXPT(rDelTime,6) + lrFun2[5] * EXPT(rDelTime,5)
    + lrFun2[6] * EXPT(rDelTime,4) + lrFun2[7] * EXPT(rDelTime,3) + lrFun2[8] * EXPT(rDelTime,2) + lrFun2[9] * rDelTime + lrFun2[10];
ELSIF rRealTime <= rNodeTime3 THEN
    rDelTime := rRealTime - rNodeTime2;
    lrFitResult := lrFun3[0] * EXPT(rDelTime,10) + lrFun3[1] * EXPT(rDelTime,9) + lrFun3[2] * EXPT(rDelTime,8) + lrFun3[3] * EXPT(rDelTime,7) + lrFun3[4] * EXPT(rDelTime,6) + lrFun3[5] * EXPT(rDelTime,5)
    + lrFun3[6] * EXPT(rDelTime,4) + lrFun3[7] * EXPT(rDelTime,3) + lrFun3[8] * EXPT(rDelTime,2) + lrFun3[9] * rDelTime + lrFun3[10];
ELSIF rRealTime <= rNodeTime4 THEN
    rDelTime := rRealTime - rNodeTime3;
    lrFitResult := lrFun4[0] * EXPT(rDelTime,10) + lrFun4[1] * EXPT(rDelTime,9) + lrFun4[2] * EXPT(rDelTime,8) + lrFun4[3] * EXPT(rDelTime,7) + lrFun4[4] * EXPT(rDelTime,6) + lrFun4[5] * EXPT(rDelTime,5)
    + lrFun4[6] * EXPT(rDelTime,4) + lrFun4[7] * EXPT(rDelTime,3) + lrFun4[8] * EXPT(rDelTime,2) + lrFun4[9] * rDelTime + lrFun4[10];
ELSIF rRealTime <= rNodeTime5 THEN
    rDelTime := rRealTime - rNodeTime4;
    lrFitResult := lrFun5[0] * EXPT(rDelTime,10) + lrFun5[1] * EXPT(rDelTime,9) + lrFun5[2] * EXPT(rDelTime,8) + lrFun5[3] * EXPT(rDelTime,7) + lrFun5[4] * EXPT(rDelTime,6) + lrFun5[5] * EXPT(rDelTime,5)
    + lrFun5[6] * EXPT(rDelTime,4) + lrFun5[7] * EXPT(rDelTime,3) + lrFun5[8] * EXPT(rDelTime,2) + lrFun5[9] * rDelTime + lrFun5[10];
ELSIF rRealTime <= rEndTime THEN
    rDelTime := rRealTime - rNodeTime5;
    lrFitResult := lrFun6[0] * EXPT(rDelTime,10) + lrFun6[1] * EXPT(rDelTime,9) + lrFun6[2] * EXPT(rDelTime,8) + lrFun6[3] * EXPT(rDelTime,7) + lrFun6[4] * EXPT(rDelTime,6) + lrFun6[5] * EXPT(rDelTime,5)
    + lrFun6[6] * EXPT(rDelTime,4) + lrFun6[7] * EXPT(rDelTime,3) + lrFun6[8] * EXPT(rDelTime,2) + lrFun6[9] * rDelTime + lrFun6[10];
ELSE
    rDelTime := rEndTime - rNodeTime5;
    lrFitResult := lrFun6[0] * EXPT(rDelTime,10) + lrFun6[1] * EXPT(rDelTime,9) + lrFun6[2] * EXPT(rDelTime,8) + lrFun6[3] * EXPT(rDelTime,7) + lrFun6[4] * EXPT(rDelTime,6) + lrFun6[5] * EXPT(rDelTime,5)
    + lrFun6[6] * EXPT(rDelTime,4) + lrFun6[7] * EXPT(rDelTime,3) + lrFun6[8] * EXPT(rDelTime,2) + lrFun6[9] * rDelTime + lrFun6[10];
END_IF

IF lrFitResult>90 THEN
	lrFitResult:=90;
ELSIF lrFitResult<3 THEN
	lrFitResult:=3;
END_IF
                  
END_FUNCTION_BLOCK

FUNCTION_BLOCK AGCMaxSearch_PB_1 //双轴静止星步进跟踪使用的代码
VAR_INPUT
	bstart:BOOL;//模块开始标识
	rAGCNow:REAL;//当前AGC值
	btrig:BOOL;//触发一次
	rStepBiasNow:REAL;//当前拉偏量 //用来判断此次搜索是否有效
	bAutoTracking:BOOL;// 自跟踪标识
	bStop:BOOL;//满足ua ue很小
	
	rCurrentPos:REAL;//当前位置
	rInterPos:REAL;//插值位置
	//rOutStepBias:REAL;//外部拉偏量
END_VAR
VAR_OUTPUT
	
	rAGCMaxBias:REAL;//输出AGC最强时的拉偏量 单位为°
	bSucess :BOOL;//数出模块是否成功
	rStepBias:REAL;//步进量
END_VAR
VAR
	ton:Standard.TON;
	rTrg:Standard.R_TRIG;//初始化上升沿检测器
	rAGCInit:REAL:=0;//初始化AGC
	rPrevAGC:REAL:=0;//上一步的AGC值 单位为V
	rBiasInit:REAL;//初始化拉偏量
	
	iCountStep:INT:=0;//计步数
	toN1: Standard.Ton;//计时器 定时触发上升沿 
	
	rDirection: INT:=1;
	rSearchNextStepTarget:REAL;//搜索当前目标位置 单位为°
	rStep:REAL:=0.0003;//步进值
	rSensitivity:REAL:=0.05;//反向灵敏度
	iCountStopMax:INT:=20;//停止计数上限
	
	rLastDirection:INT;//上一次方向，判断是否换向
	iCountDirChange:INT;//换向标识
	rAGCMaxPos:REAL;//信号最强位置
	
	rAGCLastrecord: REAL;
	iStatus: INT;
	iCountStop1:INT;//第一阶段停止标识 (正向)
	iCountStop2:INT;//(反向)
	
	rAGCMaxValue: REAL;//AGC最大值
	
	//新加的
	iCountSearchRight:INT;//搜索方向正确，提前结束标识
	
	bSearchRight:BOOL;//搜索正确标识
	//模块指行完成标识
	iCountBlockEnd:INT;//用来计数确认已达到最强位置
	iCountBlockEndMax:INT:=500;//到位计数上限
END_VAR

                    
rTrg(CLK:=bstart,Q=>);

IF rTrg.Q THEN
	rAGCInit:=rAGCNow;
	rAGCMaxValue:=rAGCNow;
	//rBiasInit:=rCurrentPos-rInterPos;//获取启动时的拉偏量
END_IF

IF bstart THEN
	//搜索换向两次
	IF iCountDirChange=2 THEN
		rSearchNextStepTarget:=rAGCMaxBias;
		IF rStepBias< rSearchNextStepTarget THEN 
			rStepBias:=rStepBias+rStep;
		ELSIF rStepBias> rSearchNextStepTarget THEN
			rStepBias:=rStepBias-rStep;
		ELSE
			rStepBias:=rStepBias;
		END_IF
		
		IF ABS((rInterPos+rStepBias)-rCurrentPos)<0.002 THEN //若位置达到最强位置，则输出成功 //可能只是路过这里,需要持续
			//需要判断稳定
			iCountBlockEnd:=iCountBlockEnd+1;
		ELSE
			iCountBlockEnd:=0;
		END_IF
		IF iCountBlockEnd>iCountBlockEndMax THEN
			iCountBlockEnd:=iCountBlockEndMax+1;
			//用TON1秒后触发
			ton(IN:=TRUE,PT:=T#1S,Q=>,ET=>);
		END_IF
		IF ton.Q THEN
			bSucess:=TRUE;
		END_IF
	ELSE
		rStepBias:=rStepBias+rDirection*rStep;
		IF rDirection<0 THEN
			//若是向小走
			IF rCurrentPos<rInterPos THEN
				IF rAGCNow<rAGCMaxValue-rSensitivity THEN
					iCountStop1:=iCountStop1+1;
					IF iCountStop1>iCountStopMax THEN
						iCountStop1:=iCountStopMax+1;
						IF bSearchRight THEN
							iCountDirChange:=2;
						ELSE
							iCountDirChange:=iCountDirChange+1;
						END_IF
						rDirection:=rDirection*(-1);
					END_IF
				ELSE
					iCountStop1:=0;	
				END_IF
				
				//新加的 测试第一阶段搜索正确后不进行第二次搜索
				IF rAGCNow>rAGCInit+rSensitivity THEN
					iCountSearchRight:=iCountSearchRight+1;
				ELSE
					iCountSearchRight:=0;
				END_IF
				IF iCountSearchRight>200 THEN
					iCountSearchRight:=201;
					bSearchRight:=TRUE;
				END_IF
				
			END_IF
		ELSE
			//若是向正走
			IF rCurrentPos>rInterPos THEN
				IF rAGCNow<rAGCMaxValue-rSensitivity THEN
					iCountStop2:=iCountStop2+1;
					IF iCountStop2>iCountStopMax THEN
						iCountStop2:=iCountStopMax+1;
						IF bSearchRight THEN
							iCountDirChange:=2;
						ELSE
							iCountDirChange:=iCountDirChange+1;
						END_IF
						rDirection:=rDirection*(-1);
					END_IF
				ELSE
					iCountStop2:=0;	
				END_IF
				
				//新加的
				IF rAGCNow>rAGCInit+rSensitivity THEN
					iCountSearchRight:=iCountSearchRight+1;
				ELSE
					iCountSearchRight:=0;
				END_IF
				IF iCountSearchRight>200 THEN
					iCountSearchRight:=201;
					bSearchRight:=TRUE;
				END_IF
				
			END_IF
		END_IF
		(*
		IF rAGCNow<rAGCInit-0.05 THEN
			iCountStop1:=iCountStop1+1;
			IF iCountStop1>150 THEN
				iCountDirChange:=iCountDirChange+1;
				rDirection:=rDirection*(-1);
			END_IF
		ELSE
			iCountStop1:=0;	
		END_IF
		*)
		
		 // 记录最强信号的拉偏量和值
		//IF rAGCNow >= rAGCInit AND rAGCNow> rAGCMaxValue THEN
		IF  rAGCNow> rAGCMaxValue THEN
			rAGCMaxBias := rStepBias;
			rAGCMaxValue := rAGCNow;
		END_IF
	END_IF
ELSE
	rStepBias:=0;
	//清空变量
	iCountDirChange:=0;
	rAGCInit:=0;
	rAGCMaxValue:=0;
	rAGCMaxBias:=0;
	rDirection:=1;
	iCountStop1:=0;
	iCountStop2:=0;
	ton(IN:=FALSE,PT:=T#1S,Q=>,ET=>);
	//rStepBias:=0;
	rSearchNextStepTarget:=0;
	bSucess:=FALSE;
	iCountSearchRight:=0;
	bSearchRight:=FALSE;
	iCountBlockEnd:=0;
END_IF


(*
IF rStepBias< rSearchNextStepTarget THEN 
	rStepBias:=rStepBias+rStep;
ELSIF rStepBias> rSearchNextStepTarget THEN
	rStepBias:=rStepBias-rStep;
ELSE
	rStepBias:=rStepBias;
END_IF*)
                  
END_FUNCTION_BLOCK

PROGRAM GPRMC_1
VAR
	com_init:gcan.FB_Com_Init;      		//gcan.FB_Com_Init为串口初始化功能块，可设定串口端口号，串口波特率等参数
	com_read:gcan.FB_Com_Read ;				//gcan.FB_Com_Read为串口接收功能块，用于通过接收串口发送给PLC的数据
	com_write:gcan.FB_Com_Write ;			//gcan.FB_Com_Write为串口发送功能块，用于发送串口数据
	m_uiError:UINT;							//用于承接功能块中报错引脚错误信息的变量
	m_out:BOOL;								//用于承接功能块中完成标志引脚数据的变量
	isFirst:BOOL:=TRUE;						//用于判断初始化只执行一次的逻辑
	mPort:BYTE;								//程序中用作设定串口端口号
	recSize:UINT;							//接收数据长度，单位：字节
	recBuf:ARRAY[0..101] OF BYTE;			//用于存放接收到的串口数据的数组
	sum_i:INT;
	checksum:BYTE;
	iYear: INT;
	iMonth: INT;
	iDay: INT;
	iHour: INT;
	iMinute: INT;
	iSecond: INT;
	strDateTimeNow : STRING;
	gnssTimestamp: ULINT;
	gnssTimestamplast:ULINT;
	icount:INT;
	high4: BYTE;
	low4: BYTE;
END_VAR
VAR_INPUT
	EN_in_1:BOOL;
END_VAR

                    ////////////////////////////////////////////////////////////////////////////////////////
//串口接收GPRMC报文解析
//日期：2024/08/25
//版本：V1.1
/////////////////////////////////////////////////////////////////////////////////////////

mPort:=1;								//串口端口号设定，GCAN-PLC-400、GCAN-PLC-510、GCAN-PLC-511，1为232，2为485
										//GCAN-PLC-324、GCAN-PLC-326，1为第一路485，2为第2路485
IF isFirst THEN
	com_init(							//串口初始化功能块
	EN_IN:=TRUE,						//串口初始化功能块使能
	xEnable:=TRUE,						//串口功能使能
	bPort:=mPort,						//串口端口号设定
	uiBaudrate:=115200,					//串口波特率设定
	bParity:=0,							//串口奇偶校验设定，0为无校验，1为奇校验，2为偶检验
	bDatabits:=8,						//数据位设定
	bStopbits:=1,						//停止位设定
	EN_OUT=>m_out,						//串口初始化功能块执行完成标志位
	uiError=>m_uiError);				//串口初始化功能块执行错误信息
	isfirst:=FALSE;						//执行一次初始化后关闭IF的条件使其之后进入ELSE程序段运行

ELSE
	
		com_read(						//串口读取功能块
		EN_in:=TRUE,					//读取功能块使能，为TRUE执行读取
		bPort:=mPort,					//串口端口号设定
		p_brxdata:=ADR(recBuf),			//读取到的串口数据引脚为指针类型，使用ADR()指向自建数组将数据存放到数组中
		uiMaxsize:=204,					//设定最大读取长度
		EN_out=>m_out,					//串口读取功能块执行完成标志位******功能块执行完成不代表接收完成********
		uiRecSize=>recSize,				//串口接收数据长度，单位：字节，大于0时说明接收到数据可用于判断是否接收
		uierror=>m_uierror);			//串口读取功能块执行错误信息
										//从数组recBuf里取数据，解析出年、月、日、时、分、秒
		//有效判定(A)+和校验(hh),前 4bit和后 4bit的 16 进制数分别以 ASCII 码表示(0~9,A~F)，高位在前。
		IF 	recBuf[0] = 36 THEN
(*			checksum := 16#00;
			FOR sum_i:=1 TO 74 BY 1 DO
				checksum:= checksum XOR recBuf[sum_i];
			END_FOR
			high4 := (SHR(checksum, 4) AND 16#0F)+16#30;
			low4 := (checksum AND 16#0F)+16#30;
			IF recBuf[76]= high4 AND recBuf[77]= low4 THEN 
*)		

			iYear:=BYTE_TO_INT(recBuf[23]-48)*1000+BYTE_TO_INT(recBuf[24]-48)*100+BYTE_TO_INT(recBuf[25]-48)*10+BYTE_TO_INT(recBuf[26]-48);
			iMonth:=BYTE_TO_INT(recBuf[20]-48)*10+BYTE_TO_INT(recBuf[21]-48);
			iDay:=BYTE_TO_INT(recBuf[17]-48)*10+BYTE_TO_INT(recBuf[18]-48);
			iHour:=BYTE_TO_INT(recBuf[7]-48)*10+BYTE_TO_INT(recBuf[8]-48)+8;
			iMinute:=BYTE_TO_INT(recBuf[9]-48)*10+BYTE_TO_INT(recBuf[10]-48);
			iSecond:=BYTE_TO_INT(recBuf[11]-48)*10+BYTE_TO_INT(recBuf[12]-48);
			
			// 计算时间戳		
			
			strDateTimeNow := CONCAT(STR1 := 'DT#', STR2 := INT_TO_STRING(iYear));
			strDateTimeNow := CONCAT(STR1 := strDateTimeNow, STR2 := '-');
			strDateTimeNow := CONCAT(STR1 := strDateTimeNow, STR2 := INT_TO_STRING(iMonth));
			strDateTimeNow := CONCAT(STR1 := strDateTimeNow, STR2 := '-');
			strDateTimeNow := CONCAT(STR1 := strDateTimeNow, STR2 := INT_TO_STRING(iDay));
			strDateTimeNow := CONCAT(STR1 := strDateTimeNow, STR2 := '-');
			strDateTimeNow := CONCAT(STR1 := strDateTimeNow, STR2 := INT_TO_STRING(iHour));
			strDateTimeNow := CONCAT(STR1 := strDateTimeNow, STR2 := ':');
			strDateTimeNow := CONCAT(STR1 := strDateTimeNow, STR2 := INT_TO_STRING(iMinute));
			strDateTimeNow := CONCAT(STR1 := strDateTimeNow, STR2 := ':');
			strDateTimeNow := CONCAT(STR1 := strDateTimeNow, STR2 := INT_TO_STRING(iSecond));
			(*
			gnssTimestamplast:=gnssTimestamp;
			
			
			*)
			gnssTimestamp := DT_TO_ULINT(TO_DT(strDateTimeNow)) * 1000;
			GVL.stGNSS_Timestap := gnssTimestamp;
		END_IF
		(*
		IF gnssTimestamplast<>gnssTimestamp THEN
			icount:=0;
		ELSE
			icount:=icount+1;
		END_IF
		*)
		


(*	IF recsize>0 THEN					//如果接收到串口数据
		
		com_write(						//串口发送功能块
		EN_IN:=TRUE,					//串口发送功能块使能，发送机制：当使能为TRUE时，PLC程序每周期运行到此处就执行一次发送
		bPort:=mPort,					//串口端口号设定
		p_bTxdata:=ADR(recbuf),			//将接收存放到数组中的数据发送出去******若发送其它数据，自建另一数组用于存放发送数据即可
		uiTxsize:=recsize,				//发送长度为接收到的数据长度******若发送其它长度，自行填写所需长度即可
		EN_OUT=>m_out,					//串口发送功能块执行完成标志位
		uierror=>m_uierror);			//串口发送功能块执行错误信息
			
	END_IF
*)	
END_IF
                  
END_PROGRAM

PROGRAM GetACUTime
VAR
    tp      : TP;           // 脉冲定时器
    toggle  : BOOL := FALSE; // 当前输出状态
    clk     : BOOL := FALSE; // 方波输出
    tick_ms : TIME := T#500MS; // 高电平/低电平持续时间
	Result : RTS_IEC_RESULT;
	stUTC_Timestamp :SYSTIME ;
	
	dRTime:ULINT;//上位机外部时间 单位ns Unix时间戳，起点是1970-1-1 0:0:0
	dModbusTime:ULINT;//Modbus临时外部时间
	iCountRemote:INT; //上位机锁定判断时间常数
	dCountRemote:ULINT;//上位机时间滑动平均常数
	dLastRTime:ULINT;//上位机上一次外部时间 单位ns Unix时间戳，起点是1970-1-1 0:0:0
	iDiffRTime:DINT;//上位机时间差值
	dDelRTime:LINT;
	dMeanDelRTime:LINT;
	rTriger:Standard.R_TRIG;//上升沿触发器
	
	iDiff:DINT;//实际时间差值
	iDiffLocal:DINT;//本地时间差值
	iDiffETime:DINT;//外部时间差值
	ulACUTimeStamp : ULINT;
END_VAR

                    
// 每次TP结束时翻转状态
IF NOT tp.Q THEN
    toggle := NOT toggle;
    tp.IN := TRUE;
    tp.PT := tick_ms;
ELSE
    tp.IN := FALSE;
END_IF

tp();

Result := SysTimeRtcHighResGet(stUTC_Timestamp);
rTriger(CLK:=toggle);
IF rTriger.Q THEN
	dRTime := modbus_slave.UTC_New;
	iDiffRTime:=ULINT_TO_DINT(dRTime-dLastRTime);
	IF ABS(iDiffRTime)>500 THEN //两次PTP时间差如果大于500毫秒,则判断为上位机时间失锁
		iCountRemote:=0;
		dCountRemote:=0;
		GVL.bRemoteTimeLock:=FALSE;
	ELSE//否则判断为上位机时间锁定并累计1分钟
		iCountRemote:=iCountRemote+1;
	END_IF
	
	IF iCountRemote>=20 THEN //累计20s认为时间可用
		iCountRemote:=20;
		dDelRTime := TO_ULINT(stUTC_Timestamp) - (dRTime + 8 * 3600 *1000);
		GVL.bRemoteTimeLock:=TRUE;
		//对外部和本机时间差做1分钟的均值滤波
	END_IF
	//GVL.dRemoteTime:=stUTC_Timestamp*1000000 - dMeanDelRTime;
	dLastRTime:=dRTime;
	(*
	IF GVL.bRemoteTimeLock THEN
		dCountRemote:= dCountRemote + 1;
		IF dCountRemote < 10000 THEN
			dMeanDelRTime := (dMeanDelRTime*(dCountRemote-1) + dDelRTime)/dCountRemote;
		ELSE
			dCountRemote := 10000;
			dMeanDelRTime := (dMeanDelRTime*(dCountRemote-1) + dDelRTime)/dCountRemote; 	
			//iDiff:=ULINT_TO_DINT(Gvl.dPTPCSTTime-dLastCSTtime);
			//dLastCSTtime:=dCSTTime;
		END_IF
	END_IF
	*)
END_IF

ulACUTimeStamp := stUTC_Timestamp - dDelRTime;
                  
END_PROGRAM

PROGRAM XPTOD_SerialCom
VAR
        com_init:gcan.FB_Com_Init;                      //gcan.FB_Com_Init为串口初始化功能块，可设定串口端口号，串口波特率等参数
        com_read:gcan.FB_Com_Read ;                                //gcan.FB_Com_Read为串口接收功能块，用于通过接收串口发送给PLC的数据
        com_write:gcan.FB_Com_Write ;                        //gcan.FB_Com_Write为串口发送功能块，用于发送串口数据
        m_uiError:UINT;                                                        //用于承接功能块中报错引脚错误信息的变量
        m_out:BOOL;                                                                //用于承接功能块中完成标志引脚数据的变量
        isFirst:BOOL:=TRUE;                                                //用于判断初始化只执行一次的逻辑
        mPort:BYTE;                                                                //程序中用作设定串口端口号
        recSize:UINT;                                                        //接收数据长度，单位：字节
        recBuf:ARRAY[0..239] OF BYTE;                        //用于存放接收到的串口数据的数组
        iYear: INT;                             //年
        iMonth: INT;                            //月
        iDay: INT;                              //日
        iHour: INT;                             //时
        iMinute: INT;                           //分
        iSecond: INT;                           //秒
    bChecksumValid: BOOL := FALSE;                //校验和
        nFrameHeadPos: INT := 0;                //帧头索引          
    nPos        : INT;                      //帧头位置
    nChecksumRx : BYTE := 0;                //和校验
        strDateTimeNow : STRING;
        gnssTimestamp: ULINT;
        gnssTimestamplast:ULINT;
        icount:INT;
END_VAR

                    ////////////////////////////////////////////////////////////////////////////////////////
//串口接收TOD报文解析
//日期：2025/05/15
//版本：V1.1
/////////////////////////////////////////////////////////////////////////////////////////

mPort:=1;                                                                //串口端口号设定，GCAN-PLC-400、GCAN-PLC-510、GCAN-PLC-511，1为232，2为485
                                                                                //GCAN-PLC-324、GCAN-PLC-326，1为第一路485，2为第2路485
IF isFirst THEN
        com_init(                                                        //串口初始化功能块
        EN_IN:=TRUE,                                                //串口初始化功能块使能
        xEnable:=TRUE,                                                //串口功能使能
        bPort:=mPort,                                                //串口端口号设定
        uiBaudrate:=115200,                                        //串口波特率设定
        bParity:=0,                                                        //串口奇偶校验设定，0为无校验，1为奇校验，2为偶检验
        bDatabits:=8,                                                //数据位设定
        bStopbits:=1,                                                //停止位设定
        EN_OUT=>m_out,                                                //串口初始化功能块执行完成标志位
        uiError=>m_uiError);                                //串口初始化功能块执行错误信息
        isfirst:=FALSE;                                                //执行一次初始化后关闭IF的条件使其之后进入ELSE程序段运行

ELSE
        
                com_read(                                                //串口读取功能块
                EN_in:=TRUE,                                        //读取功能块使能，为TRUE执行读取
                bPort:=mPort,                                        //串口端口号设定
                p_brxdata:=ADR(recBuf),                        //读取到的串口数据引脚为指针类型，使用ADR()指向自建数组将数据存放到数组中
                uiMaxsize:=240,                                        //设定最大读取长度
                EN_out=>m_out,                                        //串口读取功能块执行完成标志位******功能块执行完成不代表接收完成********
                uiRecSize=>recSize,                                //串口接收数据长度，单位：字节，大于0时说明接收到数据可用于判断是否接收
                uierror=>m_uierror);                        //串口读取功能块执行错误信息
                // 查找帧头 $X (36, 88)
                FOR nPos := 1 TO 240 DO
                        IF recBuf[nPos] = 36 AND recBuf[nPos + 1] = 88 THEN
                                nFrameHeadPos := nPos;
                                EXIT;
                        END_IF
                END_FOR
                //解析时间日期 
                IF nFrameHeadPos + 26 <= 240 THEN
                        iYear:=BYTE_TO_INT(recBuf[nFrameHeadPos+23]-48)*1000+BYTE_TO_INT(recBuf[nFrameHeadPos+24]-48)*100+BYTE_TO_INT(recBuf[nFrameHeadPos+25]-48)*10+BYTE_TO_INT(recBuf[26]-48);
                        iMonth:=BYTE_TO_INT(recBuf[nFrameHeadPos+20]-48)*10+BYTE_TO_INT(recBuf[nFrameHeadPos+21]-48);
                        iDay:=BYTE_TO_INT(recBuf[nFrameHeadPos+17]-48)*10+BYTE_TO_INT(recBuf[nFrameHeadPos+18]-48);
                        iHour:=BYTE_TO_INT(recBuf[nFrameHeadPos+7]-48)*10+BYTE_TO_INT(recBuf[nFrameHeadPos+8]-48)+8;
                        iMinute:=BYTE_TO_INT(recBuf[nFrameHeadPos+9]-48)*10+BYTE_TO_INT(recBuf[nFrameHeadPos+10]-48);
                        iSecond:=BYTE_TO_INT(recBuf[nFrameHeadPos+11]-48)*10+BYTE_TO_INT(recBuf[nFrameHeadPos+12]-48);
                        // 计算时间戳                
                        
                        strDateTimeNow := CONCAT(STR1 := 'DT#', STR2 := INT_TO_STRING(iYear));
                        strDateTimeNow := CONCAT(STR1 := strDateTimeNow, STR2 := '-');
                        strDateTimeNow := CONCAT(STR1 := strDateTimeNow, STR2 := INT_TO_STRING(iMonth));
                        strDateTimeNow := CONCAT(STR1 := strDateTimeNow, STR2 := '-');
                        strDateTimeNow := CONCAT(STR1 := strDateTimeNow, STR2 := INT_TO_STRING(iDay));
                        strDateTimeNow := CONCAT(STR1 := strDateTimeNow, STR2 := '-');
                        strDateTimeNow := CONCAT(STR1 := strDateTimeNow, STR2 := INT_TO_STRING(iHour));
                        strDateTimeNow := CONCAT(STR1 := strDateTimeNow, STR2 := ':');
                        strDateTimeNow := CONCAT(STR1 := strDateTimeNow, STR2 := INT_TO_STRING(iMinute));
                        strDateTimeNow := CONCAT(STR1 := strDateTimeNow, STR2 := ':');
                        strDateTimeNow := CONCAT(STR1 := strDateTimeNow, STR2 := INT_TO_STRING(iSecond));
                        
                        gnssTimestamplast:=gnssTimestamp;
                        gnssTimestamp := DT_TO_ULINT(TO_DT(strDateTimeNow)) * 1000;
                        GVL.stGNSS_Timestap := gnssTimestamp;                        
                END_IF
                
                IF gnssTimestamplast<>gnssTimestamp THEN
                        icount:=0;
                ELSE
                        icount:=icount+1;
                END_IF        
END_IF
                  
END_PROGRAM

PROGRAM GPRMC_1_1
VAR
        com_init:gcan.FB_Com_Init;                      //gcan.FB_Com_Init为串口初始化功能块，可设定串口端口号，串口波特率等参数
        com_read:gcan.FB_Com_Read ;                                //gcan.FB_Com_Read为串口接收功能块，用于通过接收串口发送给PLC的数据
        com_write:gcan.FB_Com_Write ;                        //gcan.FB_Com_Write为串口发送功能块，用于发送串口数据
        m_uiError:UINT;                                                        //用于承接功能块中报错引脚错误信息的变量
        m_out:BOOL;                                                                //用于承接功能块中完成标志引脚数据的变量
        isFirst:BOOL:=TRUE;                                                //用于判断初始化只执行一次的逻辑
        mPort:BYTE;                                                                //程序中用作设定串口端口号
        recSize:UINT;                                                        //接收数据长度，单位：字节
        recBuf:ARRAY[0..120] OF BYTE;                        //用于存放接收到的串口数据的数组
        iYear: INT;                             //年
        iMonth: INT;                            //月
        iDay: INT;                              //日
        iHour: INT;                             //时
        iMinute: INT;                           //分
        iSecond: INT;                           //秒
    bChecksumValid: BOOL := FALSE;                //校验和
        nFrameHeadPos: INT := 0;                //帧头索引          
    nPos        : INT;                      //帧头位置
    nChecksumRx : BYTE := 0;                //和校验
        strDateTimeNow : STRING;
        gnssTimestamp: ULINT;
        gnssTimestamplast:ULINT;
        icount:INT;
END_VAR

                    ////////////////////////////////////////////////////////////////////////////////////////
//串口接收TOD报文解析
//日期：2025/05/15
//版本：V1.1
/////////////////////////////////////////////////////////////////////////////////////////

mPort:=1;                                                                //串口端口号设定，GCAN-PLC-400、GCAN-PLC-510、GCAN-PLC-511，1为232，2为485
                                                                                //GCAN-PLC-324、GCAN-PLC-326，1为第一路485，2为第2路485
IF isFirst THEN
        com_init(                                                        //串口初始化功能块
        EN_IN:=TRUE,                                                //串口初始化功能块使能
        xEnable:=TRUE,                                                //串口功能使能
        bPort:=mPort,                                                //串口端口号设定
        uiBaudrate:=115200,                                        //串口波特率设定
        bParity:=0,                                                        //串口奇偶校验设定，0为无校验，1为奇校验，2为偶检验
        bDatabits:=8,                                                //数据位设定
        bStopbits:=1,                                                //停止位设定
        EN_OUT=>m_out,                                                //串口初始化功能块执行完成标志位
        uiError=>m_uiError);                                //串口初始化功能块执行错误信息
        isfirst:=FALSE;                                                //执行一次初始化后关闭IF的条件使其之后进入ELSE程序段运行

ELSE
        
                com_read(                                                //串口读取功能块
                EN_in:=TRUE,                                        //读取功能块使能，为TRUE执行读取
                bPort:=mPort,                                        //串口端口号设定
                p_brxdata:=ADR(recBuf),                        //读取到的串口数据引脚为指针类型，使用ADR()指向自建数组将数据存放到数组中
                uiMaxsize:=240,                                        //设定最大读取长度
                EN_out=>m_out,                                        //串口读取功能块执行完成标志位******功能块执行完成不代表接收完成********
                uiRecSize=>recSize,                                //串口接收数据长度，单位：字节，大于0时说明接收到数据可用于判断是否接收
                uierror=>m_uierror);                        //串口读取功能块执行错误信息
                // 查找帧头 $X (36, 88)
                FOR nPos := 0 TO 119 DO
                        IF recBuf[nPos] = 36 AND recBuf[nPos + 1] = 88 THEN
                                nFrameHeadPos := nPos;
                                EXIT;
                        END_IF
                END_FOR
                //解析时间日期 
                IF nFrameHeadPos + 26 <= 120 THEN
                        iYear:=BYTE_TO_INT(recBuf[nFrameHeadPos+23]-48)*1000+BYTE_TO_INT(recBuf[nFrameHeadPos+24]-48)*100+BYTE_TO_INT(recBuf[nFrameHeadPos+25]-48)*10+BYTE_TO_INT(recBuf[26]-48);
                        iMonth:=BYTE_TO_INT(recBuf[nFrameHeadPos+20]-48)*10+BYTE_TO_INT(recBuf[nFrameHeadPos+21]-48);
                        iDay:=BYTE_TO_INT(recBuf[nFrameHeadPos+17]-48)*10+BYTE_TO_INT(recBuf[nFrameHeadPos+18]-48);
                        iHour:=BYTE_TO_INT(recBuf[nFrameHeadPos+7]-48)*10+BYTE_TO_INT(recBuf[nFrameHeadPos+8]-48)+8;
                        iMinute:=BYTE_TO_INT(recBuf[nFrameHeadPos+9]-48)*10+BYTE_TO_INT(recBuf[nFrameHeadPos+10]-48);
                        iSecond:=BYTE_TO_INT(recBuf[nFrameHeadPos+11]-48)*10+BYTE_TO_INT(recBuf[nFrameHeadPos+12]-48);
                        // 计算时间戳                
                        
                        strDateTimeNow := CONCAT(STR1 := 'DT#', STR2 := INT_TO_STRING(iYear));
                        strDateTimeNow := CONCAT(STR1 := strDateTimeNow, STR2 := '-');
                        strDateTimeNow := CONCAT(STR1 := strDateTimeNow, STR2 := INT_TO_STRING(iMonth));
                        strDateTimeNow := CONCAT(STR1 := strDateTimeNow, STR2 := '-');
                        strDateTimeNow := CONCAT(STR1 := strDateTimeNow, STR2 := INT_TO_STRING(iDay));
                        strDateTimeNow := CONCAT(STR1 := strDateTimeNow, STR2 := '-');
                        strDateTimeNow := CONCAT(STR1 := strDateTimeNow, STR2 := INT_TO_STRING(iHour));
                        strDateTimeNow := CONCAT(STR1 := strDateTimeNow, STR2 := ':');
                        strDateTimeNow := CONCAT(STR1 := strDateTimeNow, STR2 := INT_TO_STRING(iMinute));
                        strDateTimeNow := CONCAT(STR1 := strDateTimeNow, STR2 := ':');
                        strDateTimeNow := CONCAT(STR1 := strDateTimeNow, STR2 := INT_TO_STRING(iSecond));
                        
                        gnssTimestamplast:=gnssTimestamp;
                        gnssTimestamp := DT_TO_ULINT(TO_DT(strDateTimeNow)) * 1000;
                        GVL.stGNSS_Timestap := gnssTimestamp;                        
                END_IF
                
                IF gnssTimestamplast<>gnssTimestamp THEN
                        icount:=0;
                ELSE
                        icount:=icount+1;
                END_IF        
END_IF
                  
END_PROGRAM

FUNCTION_BLOCK SpiralScan

VAR_INPUT
    enable : BOOL;
    delta : REAL;
    delta1 : REAL;
    n_steps : REAL;
    agc : REAL;
    locked : BOOL;
    AzError : REAL;
    ELError : REAL;
    bTrackState : BOOL;
END_VAR

VAR_OUTPUT
    azimuth : REAL;
    elevation : REAL;
    done : BOOL;
    bType : BOOL;
END_VAR

VAR
    lock_count : INT;
    best_agc : REAL;
    best_az : REAL;
    best_el : REAL;
    bInit : BOOL;
    icount0 : INT;
    icount1 : INT;
    x : REAL;
    y : REAL;
    dx : REAL;
    dy : REAL;
    step_len : REAL;
    step_count : REAL;
    segment_progress : REAL;
    move_count : REAL;
    state : INT;
    az0 : REAL;
    el0 : REAL;
    az1 : REAL;
    el1 : REAL;
    segment_az_step : REAL;
    segment_el_step : REAL;
    side_repeat : REAL;
    icountInit : INT;
    iSearchMax : INT;
    iCountSearch : INT;
    rTemp : REAL;
END_VAR

                    IF NOT enable THEN
    state := 0;
    azimuth := 0.0;
    elevation := 0.0;
    done := FALSE;
	lock_count := 0;
	icount0 := 0;
	segment_progress := 0.0;
	bInit := FALSE;
	best_agc := 0.0;
    best_az := 0.0;
    best_el := 0.0;
	icountInit := 0;
	iCountSearch := 0;
	bType := FALSE;
ELSE
    CASE state OF
        0:
			IF bTrackState THEN
				azimuth := 0.0;
				elevation := 0.0;
				done := TRUE;
				state := 3;
			ELSE
				state := 1;
				lock_count := 0;
			END_IF
        1:
            IF bTrackState THEN
				azimuth := 0.0;
				elevation := 0.0;
				done := TRUE;
				state := 3;
			ELSIF NOT bInit THEN
					x := 0.0; y := 0.0;
					dx := 1.0; dy := 0.0;
					step_len := 1.0;
					step_count := 0.0;
					move_count := 1.0;
					side_repeat := 0.0;
					az0 := 0.0; el0 := 0.0;
					az1 := delta * x;
					el1 := delta * y;
					segment_progress := 0.0;
					bInit := TRUE;
					iSearchMax := TO_INT(delta / n_steps);
					IF ABS(delta) < 1E-5 THEN
						rTemp := 0;
					ELSE
						rTemp := delta1 / delta;
					END_IF
			ELSE
					iCountSearch := iCountSearch + 1;
					IF iCountSearch <= iSearchMax THEN
						azimuth := n_steps * iCountSearch;
						elevation := n_steps * iCountSearch * rTemp;
					ELSIF iCountSearch <= 2 * iSearchMax THEN
						azimuth := delta - n_steps * (iCountSearch - iSearchMax);
						elevation := (delta - n_steps * (iCountSearch - iSearchMax)) * rTemp;
					ELSIF iCountSearch <= 3 * iSearchMax THEN
						azimuth := -1*n_steps * (iCountSearch - 2*iSearchMax);
						elevation := (-1*n_steps * (iCountSearch - 2*iSearchMax)) * rTemp;
					ELSIF iCountSearch < 4 * iSearchMax THEN
						azimuth := n_steps * (iCountSearch - 3*iSearchMax) - delta;
						elevation := (n_steps * (iCountSearch - 3*iSearchMax) - delta) * rTemp;
					END_IF

					IF ABS(delta1) < 1E-4 THEN
						elevation := 0;
					END_IF

					IF iCountSearch >= 4 * iSearchMax THEN
						azimuth := 0.0;
						elevation := 0.0;
						done := TRUE;
						state := 3;
					ELSE
						IF locked THEN
						   lock_count := lock_count + 1;
						ELSE
						   lock_count := 0;
						END_IF
						IF lock_count >= 10 THEN
						   azimuth := -Azerror;
						   elevation := -elError;
						   done := TRUE;
						   state := 2;
						END_IF
					END_IF
			END_IF
        2:
            done := TRUE;
        3:
            azimuth := 0.0;
            elevation := 0.0;
            done := TRUE;
    END_CASE

	IF state = 2 THEN
		bType := TRUE;
	ELSIF state = 3 THEN
		bType := FALSE;
	END_IF
END_IF;

                  
END_FUNCTION_BLOCK

FUNCTION_BLOCK SpiralScan_1

VAR_INPUT
    enable : BOOL;
    delta : REAL;
    n_steps : REAL;
    agc : REAL;
    locked : BOOL;
    AzError : REAL;
    ELError : REAL;
END_VAR

VAR_OUTPUT
    azimuth : REAL;
    elevation : REAL;
    done : BOOL;
    bType : BOOL;
END_VAR

VAR
    lock_count : INT;
    best_agc : REAL;
    best_az : REAL;
    best_el : REAL;
    bInit : BOOL;
    icount0 : INT;
    icount1 : INT;
    x : REAL;
    y : REAL;
    dx : REAL;
    dy : REAL;
    step_len : REAL;
    step_count : REAL;
    segment_progress : REAL;
    move_count : REAL;
    state : INT;
    az0 : REAL;
    el0 : REAL;
    az1 : REAL;
    el1 : REAL;
    segment_az_step : REAL;
    segment_el_step : REAL;
    side_repeat : REAL;
    icountInit : INT;
END_VAR

                    IF NOT enable THEN
    state := 0;
    azimuth := 0.0;
    elevation := 0.0;
    done := FALSE;
	lock_count := 0;
	icount0 := 0;
	segment_progress := 0.0;
	bInit := FALSE;
	best_agc := 0.0;
    best_az := 0.0;
    best_el := 0.0;
	icountInit := 0;
	bType := FALSE;
ELSE
    CASE state OF
        0:
			state := 1;
			lock_count := 0;
        1:
            IF NOT bInit THEN
				x := 0.0; y := 0.0;
				dx := 1.0; dy := 0.0;
				step_len := 1.0;
				step_count := 0.0;
				move_count := 1.0;
				side_repeat := 0.0;
				az0 := 0.0; el0 := 0.0;
				az1 := delta * x;
				el1 := delta * y;
				segment_az_step := (az1 - az0) / n_steps;
				segment_el_step := (el1 - el0) / n_steps;
				segment_progress := 0.0;
				bInit := TRUE;
			ELSE
				azimuth := az0 + segment_az_step * (segment_progress + 1.0);
				elevation := el0 + segment_el_step * (segment_progress + 1.0);
				segment_progress := segment_progress + 1.0;

				IF segment_progress >= n_steps THEN
					segment_progress := 0.0;
					az0 := az1;
					el0 := el1;
					x := x + dx;
					y := y + dy;
					move_count := move_count + 1.0;

					az1 := delta * x;
					el1 := delta * y;
					segment_az_step := (az1 - az0) / n_steps;
					segment_el_step := (el1 - el0) / n_steps;

					step_count := step_count + 1.0;
					IF step_count >= step_len THEN
						step_count := 0.0;
						IF dx = 1.0 AND dy = 0.0 THEN
							dx := 0.0; dy := 1.0;
						ELSIF dx = 0.0 AND dy = 1.0 THEN
							dx := -1.0; dy := 0.0;
						ELSIF dx = -1.0 AND dy = 0.0 THEN
							dx := 0.0; dy := -1.0;
						ELSIF dx = 0.0 AND dy = -1.0 THEN
							dx := 1.0; dy := 0.0;
						END_IF

						side_repeat := side_repeat + 1.0;
						IF side_repeat >= 2.0 THEN
							side_repeat := 0.0;
							step_len := step_len + 1.0;
						END_IF
					END_IF
				END_IF

				IF ABS(azimuth - 4 * delta) < 1E-6 AND ABS(elevation) < 1E-6 THEN
					azimuth := 0.0;
					elevation := 0.0;
					done := TRUE;
					state := 3;
				ELSE
					IF locked THEN
					   lock_count := lock_count + 1;
					ELSE
					   lock_count := 0;
					END_IF
					IF lock_count >= 10 THEN
					   azimuth := -Azerror;
            		   elevation := -elError;
					   done := TRUE;
					   state := 2;
					END_IF
				END_IF
			END_IF
        2:
            done := TRUE;
        3:
            azimuth := 0.0;
            elevation := 0.0;
            done := TRUE;
    END_CASE
	IF state = 2 THEN
		bType := TRUE;
	ELSIF state = 3 THEN
		bType := FALSE;
	END_IF
END_IF;

                  
END_FUNCTION_BLOCK

FUNCTION_BLOCK FB_PhaseFit
(* Offline candidate. Feed ONE coherent, validated sample per xSample pulse.
   Coordinates: positive Az=right, positive El=up. Desired response is -I.
   eAz/eEl must already have consistent signed engineering units.
   Do not subtract 2.5 from the existing signed serial values without protocol proof. *)
VAR_INPUT
    xReset : BOOL;
    xSample : BOOL;
    xFinish : BOOL;
    lrAz : LREAL;
    lrEl : LREAL;
    lrUa : LREAL;
    lrUe : LREAL;
    lrCurrentPhaseDeg : LREAL;
    (* +1: increasing hardware phase rotates measured response CCW; -1: CW; 0: unknown *)
    iPhaseDirection : INT;
END_VAR
VAR_OUTPUT
    xFitValid : BOOL;
    xSuggestedValid : BOOL;
    uiError : UINT;
    udiSamples : UDINT;
    lrKaa, lrKae, lrKea, lrKee : LREAL;
    lrInterceptAz, lrInterceptEl : LREAL;
    lrResponseAngleDeg : LREAL;
    lrCorrectionDeg, lrSuggestedDeg : LREAL;
    lrCandidatePlusDeg, lrCandidateMinusDeg : LREAL;
    lrOrthErrorDeg : LREAL;
    lrResidualAz, lrResidualEl : LREAL;
    lrCrossAz, lrCrossEl : LREAL;
END_VAR
VAR
    sx, sy, su, sv, sxx, syy, sxy, sxu, syu, sxv, syv, suu, svv : LREAL;
    n, xx, yy, xy, xu, yu, xv, yv, uu, vv, det : LREAL;
    ga, ge, dot, a, b, phi, pi, base, sse : LREAL;
    finishOld : BOOL;
END_VAR

                    pi := 3.141592653589793;
IF xReset THEN
    sx:=0; sy:=0; su:=0; sv:=0; sxx:=0; syy:=0; sxy:=0;
    sxu:=0; syu:=0; sxv:=0; syv:=0; suu:=0; svv:=0;
    udiSamples:=0; uiError:=0; xFitValid:=FALSE; xSuggestedValid:=FALSE;
    lrKaa:=0; lrKae:=0; lrKea:=0; lrKee:=0;
    lrInterceptAz:=0; lrInterceptEl:=0; lrResponseAngleDeg:=0;
    lrCorrectionDeg:=0; lrSuggestedDeg:=0;
    lrCandidatePlusDeg:=0; lrCandidateMinusDeg:=0;
    lrOrthErrorDeg:=0; lrResidualAz:=0; lrResidualEl:=0;
    lrCrossAz:=0; lrCrossEl:=0;
ELSIF xSample AND NOT xFinish THEN
    IF udiSamples < 100000 THEN
        udiSamples:=udiSamples+1;
        sx:=sx+lrAz; sy:=sy+lrEl; su:=su+lrUa; sv:=sv+lrUe;
        sxx:=sxx+lrAz*lrAz; syy:=syy+lrEl*lrEl; sxy:=sxy+lrAz*lrEl;
        sxu:=sxu+lrAz*lrUa; syu:=syu+lrEl*lrUa;
        sxv:=sxv+lrAz*lrUe; syv:=syv+lrEl*lrUe;
        suu:=suu+lrUa*lrUa; svv:=svv+lrUe*lrUe;
    ELSE
        uiError:=1;
    END_IF;
END_IF;

IF xFinish AND NOT finishOld AND NOT xReset THEN
    xFitValid:=FALSE; xSuggestedValid:=FALSE;
    IF udiSamples < 30 OR uiError <> 0 THEN
        uiError:=2;
    ELSE
        n:=UDINT_TO_LREAL(udiSamples);
        xx:=sxx-sx*sx/n; yy:=syy-sy*sy/n; xy:=sxy-sx*sy/n;
        xu:=sxu-sx*su/n; yu:=syu-sy*su/n;
        xv:=sxv-sx*sv/n; yv:=syv-sy*sv/n;
        uu:=suu-su*su/n; vv:=svv-sv*sv/n;
        det:=xx*yy-xy*xy;
        IF xx <= 1E-12 OR yy <= 1E-12 OR det <= 0.01*xx*yy THEN
            uiError:=3; (* insufficient two-axis excitation *)
        ELSE
            lrKaa:=(xu*yy-yu*xy)/det;
            lrKae:=(yu*xx-xu*xy)/det;
            lrKea:=(xv*yy-yv*xy)/det;
            lrKee:=(yv*xx-xv*xy)/det;
            lrInterceptAz:=(su-lrKaa*sx-lrKae*sy)/n;
            lrInterceptEl:=(sv-lrKea*sx-lrKee*sy)/n;
            ga:=SQRT(lrKaa*lrKaa+lrKea*lrKea);
            ge:=SQRT(lrKae*lrKae+lrKee*lrKee);
            sse:=MAX(0.0,uu-lrKaa*xu-lrKae*yu);
            lrResidualAz:=SQRT(sse/n);
            sse:=MAX(0.0,vv-lrKea*xv-lrKee*yv);
            lrResidualEl:=SQRT(sse/n);
            IF ga < 1E-6 OR ge < 1E-6 OR (uu+vv) < 1E-10 THEN
                uiError:=4; (* no usable response *)
            ELSIF (lrKaa*lrKee-lrKae*lrKea) <= 0 THEN
                uiError:=5; (* reflection/polarity mismatch; common rotation cannot fix *)
            ELSE
                dot:=(lrKaa*lrKae+lrKea*lrKee)/(ga*ge);
                dot:=LIMIT(-1.0,dot,1.0);
                lrOrthErrorDeg:=ABS(90.0-ACOS(dot)*180.0/pi);
                (* Normalize columns to prevent unequal axis gains dominating angle.
                   For M=R(phi)*diag(-ga,-ge), a=2*cos(phi), b=2*sin(phi). *)
                a:=-lrKaa/ga-lrKee/ge;
                b:=-lrKea/ga+lrKae/ge;
                IF ABS(a)+ABS(b)<1E-9 THEN
                    uiError:=6;
                ELSE
                    IF ABS(a)<1E-12 THEN
                        IF b>=0 THEN phi:=pi/2; ELSE phi:=-pi/2; END_IF;
                    ELSE
                        phi:=ATAN(b/a);
                        IF a<0 THEN
                            IF b>=0 THEN phi:=phi+pi; ELSE phi:=phi-pi; END_IF;
                        END_IF;
                    END_IF;
                    lrResponseAngleDeg:=phi*180.0/pi;
                    (* Finite diagnostic ratio; 1E6 means a vanishing main channel. *)
                    lrCrossAz:=ABS(lrKea)/MAX(ABS(lrKaa),ga*1E-6);
                    lrCrossEl:=ABS(lrKae)/MAX(ABS(lrKee),ge*1E-6);
                    IF lrOrthErrorDeg>10.0 OR
                       (lrResidualAz*lrResidualAz+lrResidualEl*lrResidualEl)*n > 0.1*(uu+vv) THEN
                        uiError:=7; (* diagnostic fit retained, correction rejected *)
                    ELSIF lrCurrentPhaseDeg<0 OR lrCurrentPhaseDeg>360 THEN
                        uiError:=8;
                    ELSE
                        xFitValid:=TRUE;
                        base:=lrCurrentPhaseDeg;
                        lrCandidatePlusDeg:=base+lrResponseAngleDeg;
                        lrCandidateMinusDeg:=base-lrResponseAngleDeg;
                        IF lrCandidatePlusDeg<0 THEN lrCandidatePlusDeg:=lrCandidatePlusDeg+360; END_IF;
                        IF lrCandidatePlusDeg>=360 THEN lrCandidatePlusDeg:=lrCandidatePlusDeg-360; END_IF;
                        IF lrCandidateMinusDeg<0 THEN lrCandidateMinusDeg:=lrCandidateMinusDeg+360; END_IF;
                        IF lrCandidateMinusDeg>=360 THEN lrCandidateMinusDeg:=lrCandidateMinusDeg-360; END_IF;
                        IF iPhaseDirection=1 OR iPhaseDirection=-1 THEN
                            lrCorrectionDeg:=-lrResponseAngleDeg/INT_TO_LREAL(iPhaseDirection);
                            lrSuggestedDeg:=base+lrCorrectionDeg;
                            IF lrSuggestedDeg<0 THEN lrSuggestedDeg:=lrSuggestedDeg+360; END_IF;
                            IF lrSuggestedDeg>=360 THEN lrSuggestedDeg:=lrSuggestedDeg-360; END_IF;
                            xSuggestedValid:=TRUE;
                        END_IF;
                    END_IF;
                END_IF;
            END_IF;
        END_IF;
    END_IF;
END_IF;
finishOld:=xFinish AND NOT xReset;
                  
END_FUNCTION_BLOCK

FUNCTION_BLOCK FB_PhaseTriangle
(* Pure offset generator. Does NOT write axis commands or change operating modes.
   Caller supplies elapsed seconds and motion permission; xStart is rising-edge.
   xAbort returns offsets smoothly while permission remains valid.
   Permission loss holds offsets and sets xFault: existing axis safety owns stopping.
   Release a held offset only after the caller has safely transferred command ownership. *)
VAR_INPUT
    xStart, xAbort, xPermit : BOOL;
    xResetHeld : BOOL;
    lrDtSec : LREAL;
    lrRadiusDeg : LREAL := 0.05;
    lrLegTimeSec : LREAL := 10.0;
    lrSettleSec : LREAL := 1.0;
END_VAR
VAR_OUTPUT
    xBusy, xDone, xAborted, xFault : BOOL;
    uiState : UINT;
    lrAzBias, lrElBias : LREAL;
    xCollect : BOOL;
END_VAR
VAR
    startOld : BOOL;
    elapsed, leg, settle, side, u, blend : LREAL;
    fromAz, fromEl, toAz, toEl : LREAL;
END_VAR

                    xCollect:=FALSE;
IF xResetHeld AND NOT xPermit AND uiState=900 THEN
    uiState:=0; xBusy:=FALSE; xFault:=FALSE;
    lrAzBias:=0; lrElBias:=0;
END_IF;
IF xStart AND NOT startOld AND NOT xBusy AND uiState<>900 THEN
    xDone:=FALSE; xAborted:=FALSE; xFault:=FALSE;
    (* 0.1 is an unvalidated commissioning ceiling, NOT a proven linear range. *)
    IF NOT xPermit OR lrRadiusDeg<=0 OR lrRadiusDeg>0.1 OR
       lrLegTimeSec<2 OR lrSettleSec<0.1 OR lrSettleSec>30 THEN
        xFault:=TRUE;
    ELSE
        side:=lrRadiusDeg/SQRT(2.0);
        leg:=lrLegTimeSec; settle:=lrSettleSec;
        elapsed:=0; lrAzBias:=0; lrElBias:=0;
        uiState:=10; xBusy:=TRUE;
    END_IF;
END_IF;
startOld:=xStart;

IF xBusy AND uiState<>900 THEN
    IF NOT xPermit OR lrDtSec<=0 OR lrDtSec>0.1 THEN
        xFault:=TRUE; uiState:=900;
    ELSE
        IF xAbort AND uiState<>800 THEN
            fromAz:=lrAzBias; fromEl:=lrElBias;
            toAz:=0; toEl:=0; elapsed:=0;
            xAborted:=TRUE; uiState:=800;
        END_IF;
        elapsed:=elapsed+lrDtSec;
        CASE uiState OF
            10,30,50,70:
                xCollect:=TRUE; (* caller still gates new-frame, quality, position settling *)
                IF elapsed>=settle THEN
                    elapsed:=0; fromAz:=lrAzBias; fromEl:=lrElBias;
                    CASE uiState OF
                        10: toAz:=0; toEl:=side; uiState:=20;
                        30: toAz:=side; toEl:=side; uiState:=40;
                        50: toAz:=0; toEl:=0; uiState:=60;
                        70: xBusy:=FALSE; xDone:=TRUE; uiState:=0;
                    END_CASE;
                END_IF;
            20,40,60,800:
                u:=LIMIT(0.0,elapsed/leg,1.0);
                blend:=u*u*u*(10.0+u*(-15.0+6.0*u));
                lrAzBias:=fromAz+(toAz-fromAz)*blend;
                lrElBias:=fromEl+(toEl-fromEl)*blend;
                xCollect:=(uiState<>800) AND (u>0.1) AND (u<0.9);
                IF u>=1 THEN
                    elapsed:=0;
                    IF uiState=800 THEN
                        xBusy:=FALSE; uiState:=0;
                    ELSE
                        uiState:=uiState+10;
                    END_IF;
                END_IF;
        END_CASE;
    END_IF;
END_IF;
                  
END_FUNCTION_BLOCK

PROGRAM PRG_PhaseCalibration
(* Called ONLY at the end of SecurityCheck, once per Canopen 10 ms cycle.
   Fixed position mode only. No writes to modes, enables, tracking or persistence.
   Loss of ownership gives command control back to the existing program immediately.
   This is not an emergency-stop/safety function. *)
VAR
    path : FB_PhaseTriangle;
    fit : FB_PhaseFit;
    startOld, startPulse, accepted, permit, ownership, quality : BOOL;
    sample, finish, newRx, rxLock, doneOld, abortRun : BOOL;
    seq, lastSeq : UDINT;
    age : LREAL := 999;
    sampleTime : LREAL;
    ua, ue, eb, az, el, centerAz, centerEl : LREAL;
    baseAz, baseEl, phase, minEb : LREAL;
    direction : INT;
END_VAR

                    startPulse:=GVL_PhaseCal.xStart AND NOT startOld;
startOld:=GVL_PhaseCal.xStart;
accepted:=FALSE; sample:=FALSE; newRx:=FALSE;
age:=MIN(age+0.01,999.0);
sampleTime:=MIN(sampleTime+0.01,1.0);
seq:=GVL_PhaseCal.udiRxSeq;
IF seq<>lastSeq AND seq MOD 2=0 THEN
    ua:=GVL_PhaseCal.lrRxUa; ue:=GVL_PhaseCal.lrRxUe;
    eb:=GVL_PhaseCal.lrRxEbN0;
    az:=GVL_PhaseCal.lrRxAz; el:=GVL_PhaseCal.lrRxEl;
    rxLock:=GVL_PhaseCal.xRxLock;
    IF seq=GVL_PhaseCal.udiRxSeq THEN
        lastSeq:=seq; age:=0; newRx:=TRUE;
    END_IF;
END_IF;

ownership:=NOT GVL.bLocalCtrl AND GVL.Axis1Remote.iMode=2 AND
    GVL.Axis2Remote.iMode=2 AND NOT GVL.bStartTrack AND
    NOT GVL.bStartLocalAutoTrack AND NOT Modbus_Slave.bStartTrackAcu AND
    NOT Modbus_Slave.bSearch AND NOT SecurityCheck.bScanRun AND
    ABS(SecurityCheck.aztest)<0.00001 AND ABS(SecurityCheck.eltest)<0.00001;
permit:=ownership AND GVL.Axis1Status.bServo_Enable AND
    GVL.Axis2Status.bServo_Enable AND NOT GVL.Axis1Status.Error AND
    NOT GVL.Axis2Status.Error AND NOT GVL.Axis1Status.ErrorStop AND
    NOT GVL.Axis2Status.ErrorStop AND GVL.eAzErrorcode=0 AND GVL.eElErrorcode=0 AND
    NOT SecurityCheck.bPrelimit_1 AND NOT SecurityCheck.bPrelimit_2 AND
    NOT SecurityCheck.bFinallimit_1 AND NOT SecurityCheck.bFinallimit_2;
IF path.xBusy THEN
    (* Never mask a changed ACU target by holding the old calibration center. *)
    permit:=permit AND ABS(REAL_TO_LREAL(Modbus_Slave.rPosCmd_2)-baseAz)<0.00001 AND
        ABS(REAL_TO_LREAL(Modbus_Slave.rPosCmd_1)-baseEl)<0.00001;
END_IF;
quality:=age<0.3 AND rxLock AND ABS(ua)<4.5 AND ABS(ue)<4.5 AND
    GVL_PhaseCal.uiSerialError=0 AND GVL_PhaseCal.xRxAlignmentConfirmed;
GVL_PhaseCal.xReady:=permit AND quality AND eb>=GVL_PhaseCal.lrMinEbN0 AND
    NOT path.xBusy AND NOT GVL_PhaseCal.xFault AND NOT GVL_PhaseCal.xAbort AND
    ABS(REAL_TO_LREAL(GVL.rFctPosReal_2)-REAL_TO_LREAL(Modbus_Slave.rPosCmd_2))<0.01 AND
    ABS(REAL_TO_LREAL(GVL.rFctPosReal_1)-REAL_TO_LREAL(Modbus_Slave.rPosCmd_1))<0.01 AND
    ABS(REAL_TO_LREAL(Modbus_Slave.rPosCmd_2))<274.8 AND
    Modbus_Slave.rPosCmd_1>93.2 AND Modbus_Slave.rPosCmd_1<179.8;

IF GVL_PhaseCal.xReset AND NOT path.xBusy THEN
    GVL_PhaseCal.xFault:=FALSE; GVL_PhaseCal.uiError:=0;
END_IF;
IF startPulse AND NOT path.xBusy THEN
    GVL_PhaseCal.xDone:=FALSE;
    GVL_PhaseCal.xFitValid:=FALSE; GVL_PhaseCal.xSuggestedValid:=FALSE;
    IF NOT GVL_PhaseCal.xReady OR GVL_PhaseCal.lrCurrentPhaseDeg<0 OR
       GVL_PhaseCal.lrCurrentPhaseDeg>360 OR GVL_PhaseCal.lrMinEbN0<0 OR
       GVL_PhaseCal.lrRadiusDeg<=0 OR GVL_PhaseCal.lrRadiusDeg>0.1 OR
       GVL_PhaseCal.lrLegTimeSec<2 OR GVL_PhaseCal.lrLegTimeSec>60 OR
       GVL_PhaseCal.lrSettleSec<0.1 OR GVL_PhaseCal.lrSettleSec>30 THEN
        GVL_PhaseCal.uiError:=10; GVL_PhaseCal.xFault:=TRUE;
    ELSE
        baseAz:=REAL_TO_LREAL(Modbus_Slave.rPosCmd_2);
        baseEl:=REAL_TO_LREAL(Modbus_Slave.rPosCmd_1);
        centerAz:=-baseAz; centerEl:=baseEl-90;
        phase:=GVL_PhaseCal.lrCurrentPhaseDeg;
        direction:=GVL_PhaseCal.iPhaseDirection; minEb:=GVL_PhaseCal.lrMinEbN0;
        accepted:=TRUE; sampleTime:=0;
        GVL_PhaseCal.uiError:=0; GVL_PhaseCal.xFault:=FALSE;
    END_IF;
END_IF;

abortRun:=GVL_PhaseCal.xAbort;
IF path.xBusy AND path.uiState<>800 AND path.uiState<>900 THEN
    IF NOT quality OR eb<minEb THEN
        abortRun:=TRUE; GVL_PhaseCal.uiError:=20; GVL_PhaseCal.xFault:=TRUE;
    END_IF;
    IF ABS(-REAL_TO_LREAL(GVL.rFctPosReal_2)-centerAz-path.lrAzBias)>0.1 OR
       ABS(REAL_TO_LREAL(GVL.rFctPosReal_1)-90-centerEl-path.lrElBias)>0.1 THEN
        abortRun:=TRUE; GVL_PhaseCal.uiError:=21; GVL_PhaseCal.xFault:=TRUE;
    END_IF;
END_IF;
path(xStart:=accepted, xAbort:=abortRun, xPermit:=permit,
    xResetHeld:=GVL_PhaseCal.xReset AND NOT GVL.Axis1Status.bServo_Enable AND
        NOT GVL.Axis2Status.bServo_Enable,
    lrDtSec:=0.01, lrRadiusDeg:=GVL_PhaseCal.lrRadiusDeg,
    lrLegTimeSec:=GVL_PhaseCal.lrLegTimeSec, lrSettleSec:=GVL_PhaseCal.lrSettleSec);
IF path.xFault THEN
    GVL_PhaseCal.xFault:=TRUE; GVL_PhaseCal.uiError:=22;
END_IF;
IF path.xBusy AND permit AND path.uiState<>900 THEN
    (* Same signs as existing eltest/aztest target offsets. *)
    GVL.Axis1Remote.rPosCmd:=LREAL_TO_REAL(baseEl+path.lrElBias);
    GVL.Axis2Remote.rPosCmd:=LREAL_TO_REAL(baseAz-path.lrAzBias);
END_IF;
IF path.xBusy AND path.xCollect AND quality AND eb>=minEb AND
   newRx AND sampleTime>=0.05 AND NOT GVL_PhaseCal.xFault AND NOT path.xAborted THEN
    sample:=TRUE; sampleTime:=0;
END_IF;
finish:=path.xDone AND NOT doneOld AND NOT GVL_PhaseCal.xFault;
IF finish AND (ABS(-REAL_TO_LREAL(GVL.rFctPosReal_2)-centerAz)>0.01 OR
              ABS(REAL_TO_LREAL(GVL.rFctPosReal_1)-90-centerEl)>0.01) THEN
    finish:=FALSE; GVL_PhaseCal.xFault:=TRUE; GVL_PhaseCal.uiError:=31;
END_IF;
doneOld:=path.xDone;
fit(xReset:=accepted, xSample:=sample, xFinish:=finish,
    lrAz:=az-centerAz, lrEl:=el-centerEl, lrUa:=ua, lrUe:=ue,
    lrCurrentPhaseDeg:=phase, iPhaseDirection:=direction);
IF finish THEN
    GVL_PhaseCal.xDone:=TRUE;
    GVL_PhaseCal.xFitValid:=fit.xFitValid;
    GVL_PhaseCal.xSuggestedValid:=fit.xSuggestedValid;
    IF NOT fit.xFitValid THEN
        GVL_PhaseCal.xFault:=TRUE; GVL_PhaseCal.uiError:=30;
    END_IF;
END_IF;
GVL_PhaseCal.xBusy:=path.xBusy; GVL_PhaseCal.xAborted:=path.xAborted;
GVL_PhaseCal.uiState:=path.uiState; GVL_PhaseCal.uiFitError:=fit.uiError;
GVL_PhaseCal.lrAzBias:=path.lrAzBias; GVL_PhaseCal.lrElBias:=path.lrElBias;
GVL_PhaseCal.lrRxAgeSec:=age; GVL_PhaseCal.udiSamples:=fit.udiSamples;
GVL_PhaseCal.lrResponseAngleDeg:=fit.lrResponseAngleDeg;
GVL_PhaseCal.lrCorrectionDeg:=fit.lrCorrectionDeg;
GVL_PhaseCal.lrSuggestedDeg:=fit.lrSuggestedDeg;
GVL_PhaseCal.lrCandidatePlusDeg:=fit.lrCandidatePlusDeg;
GVL_PhaseCal.lrCandidateMinusDeg:=fit.lrCandidateMinusDeg;
GVL_PhaseCal.lrOrthErrorDeg:=fit.lrOrthErrorDeg;
GVL_PhaseCal.lrResidualAz:=fit.lrResidualAz; GVL_PhaseCal.lrResidualEl:=fit.lrResidualEl;
GVL_PhaseCal.lrKaa:=fit.lrKaa; GVL_PhaseCal.lrKae:=fit.lrKae;
GVL_PhaseCal.lrKea:=fit.lrKea; GVL_PhaseCal.lrKee:=fit.lrKee;
                  
END_PROGRAM

CONFIGURATION Device
  RESOURCE Application ON PLC
(* global variable list GVL *)
VAR_GLOBAL
    bElCtrlBit0 AT %QX4.0 : BOOL;
    bElCtrlBit1 AT %QX4.1 : BOOL;
    bElCtrlBit2 AT %QX4.2 : BOOL;
    bElCtrlBit3 AT %QX4.3 : BOOL;
    bElCtrlBit4 AT %QX4.4 : BOOL;
    bElCtrlBit5 AT %QX4.5 : BOOL;
    bElCtrlBit7 AT %QX4.7 : BOOL;
    bElCtrlBit8 AT %QX5.0 : BOOL;
    diElTargetVel AT %QD2 : DINT;
    diElTargetPos AT %QD3 : DINT;
    diElTargetAcc AT %QD4 : UDINT;
    diElTargetDec AT %QD5 : UDINT;
    bElStsBit0 AT %IX4.0 : BOOL;
    bElStsBit1 AT %IX4.1 : BOOL;
    bElStsBit2 AT %IX4.2 : BOOL;
    bElStsBit3 AT %IX4.3 : BOOL;
    bElStsBit10 AT %IX5.2 : BOOL;
    bElStsBit12 AT %IX5.4 : BOOL;
    diElActVel AT %ID2 : DINT;
    diElActPos AT %ID3 : DINT;
    siElMode AT %QB6 : UINT;
    eElErrorcode AT %IW3 : UINT;
    bAzCtrlBit0 AT %QX24.0 : BOOL;
    bAzCtrlBit1 AT %QX24.1 : BOOL;
    bAzCtrlBit2 AT %QX24.2 : BOOL;
    bAzCtrlBit3 AT %QX24.3 : BOOL;
    bAzCtrlBit4 AT %QX24.4 : BOOL;
    bAzCtrlBit5 AT %QX24.5 : BOOL;
    bAzCtrlBit7 AT %QX24.7 : BOOL;
    bAzCtrlBit8 AT %QX25.0 : BOOL;
    diAzTargetVel AT %QD7 : DINT;
    diAzTargetPos AT %QD8 : DINT;
    diAzTargetAcc AT %QD9 : UDINT;
    diAzTargetDec AT %QD10 : UDINT;
    bAzStsBit0 AT %IX24.0 : BOOL;
    bAzStsBit1 AT %IX24.1 : BOOL;
    bAzStsBit2 AT %IX24.2 : BOOL;
    bAzStsBit3 AT %IX24.3 : BOOL;
    bAzStsBit10 AT %IX25.2 : BOOL;
    bAzStsBit12 AT %IX25.4 : BOOL;
    diAzActVel AT %ID7 : DINT;
    diAzActPos AT %ID8 : DINT;
    siAzMode AT %QB26 : UINT;
    eAzErrorcode AT %IW13 : UINT;
    bTiCtrlBit0 AT %QX44.0 : BOOL;
    bTiCtrlBit1 AT %QX44.1 : BOOL;
    bTiCtrlBit2 AT %QX44.2 : BOOL;
    bTiCtrlBit3 AT %QX44.3 : BOOL;
    bTiCtrlBit4 AT %QX44.4 : BOOL;
    bTiCtrlBit5 AT %QX44.5 : BOOL;
    bTiCtrlBit7 AT %QX44.7 : BOOL;
    bTiCtrlBit8 AT %QX45.0 : BOOL;
    diTiTargetVel AT %QD12 : DINT;
    diTiTargetPos AT %QD13 : DINT;
    diTiTargetAcc AT %QD14 : UDINT;
    diTiTargetDec AT %QD15 : UDINT;
    bTiStsBit0 AT %IX44.0 : BOOL;
    bTiStsBit1 AT %IX44.1 : BOOL;
    bTiStsBit2 AT %IX44.2 : BOOL;
    bTiStsBit3 AT %IX44.3 : BOOL;
    bTiStsBit10 AT %IX45.2 : BOOL;
    bTiStsBit12 AT %IX45.4 : BOOL;
    diTiActVel AT %ID12 : DINT;
    diTiActPos AT %ID13 : DINT;
    siTiMode AT %QB46 : UINT;
    eTiErrorcode AT %IW23 : UINT;
    dDelTime : DINT;
    stGNSS_Timestap : ULINT;
    dRealTime : ULINT;
    bLocalCtrl : BOOL;
    bError_Reset : BOOL;
    Error_code : INT;
    Axis1Local : AxisCrtlStruct;
    Axis1Remote : AxisCrtlStruct;
    Axis1Status : AxisStatus;
    Axis1Visible : AxisVisible;
    rFctPosReal_1 : LREAL;
    rFctVelReal_1 : LREAL;
    rFctAccReal_1 : LREAL;
    rFctDecReal_1 : LREAL;
    Axis2Local : AxisCrtlStruct;
    Axis2Remote : AxisCrtlStruct;
    Axis2Status : AxisStatus;
    Axis2Visible : AxisVisible;
    rFctPosReal_2 : REAL;
    rFctVelReal_2 : LREAL;
    rFctAccReal_2 : LREAL;
    rFctDecReal_2 : LREAL;
    Axis3Local : AxisCrtlStruct;
    Axis3Remote : AxisCrtlStruct;
    Axis3Status : AxisStatus;
    Axis3Visible : AxisVisible;
    rFctPosReal_3 : REAL;
    rFctVelReal_3 : LREAL;
    rFctAccReal_3 : LREAL;
    rFctDecReal_3 : LREAL;
    bStartTrack : BOOL;
    Chan1AGC : REAL;
    Chan1Ua : REAL;
    Chan1Ue : REAL;
    Chan1Lock : BOOL;
    Chan1Online : BOOL;
    Chan2AGC : REAL;
    Chan2Ua : REAL;
    Chan2Ue : REAL;
    Chan2Lock : BOOL;
    Chan2Online : BOOL;
    Chanthreshold : REAL;
    AzV : AxisCrtlStruct;
    ElV : AxisCrtlStruct;
    TiV : AxisCrtlStruct;
    iTest : INT;
    a : INT;
    iVisualSwitch : INT;
    bAzVisable : BOOL;
    bElVisable : BOOL;
    bTlVisable : BOOL;
    bLocalAutoTrackVis : BOOL;
    bStartLocalAutoTrack : BOOL;
    bRemoteTimeLock : BOOL;
    Ti : REAL;
    El : REAL;
    bTimeSwich : BOOL;
    rvAzKpBase : REAL := 1;
    rvAzKiBase : REAL := 0.01;
    rvAzKpscale : REAL := 0.01;
    rvAzKiscale : REAL := 0.01;
    rvElKpBase : REAL := 1;
    rvElKiBase : REAL := 0.01;
    rvElKpscale : REAL := 0.01;
    rvElKiscale : REAL := 0.01;
    rvAzKpMax : REAL := 1;
    rvAzKiMax : REAL := 0.01;
    rvElKpMax : REAL := 1;
    rvElKiMax : REAL := 0.01;
    rvAzThre : REAL := 10.0;
    rvElThre : REAL := 10.0;
    bTrackingModeTemp : BOOL := FALSE; // 0 ACU转自跟踪；1 自己转
    rAzScanRangeTemp : REAL := 0.3;
    rElScanRangeTemp : REAL := 0;
    rErrorTherTemp : REAL := 3.0;
    rStepTemp : REAL := 0.0015;
    rEbN0LockThreEdit : REAL := 20.0; // 可视化编辑，写入 PersistentVars.rEbN0LockThre
END_VAR
(* global variable list PersistentVars *)
{attribute 'qualified_only'}
VAR_GLOBAL
    TiOffset : REAL := 0;
    ElOffset : REAL := 0;
    rAzKpBase : REAL := 0.9;
    rAzKiBase : REAL := 0.009;
    rAzKpscale : REAL := 0.02;
    rAzKiscale : REAL := 0.002;
    rElKpBase : REAL := 1;
    rElKiBase : REAL := 0.01;
    rElKpscale : REAL := 0.01;
    rElKiscale : REAL := 0.001;
    rAzKpMax : REAL := 2.5;
    rAzKiMax : REAL := 0.03;
    rElKpMax : REAL := 1.5;
    rElKiMax : REAL := 0.03;
    rAzThre : REAL := 80.0;
    rElThre : REAL := 80.0;
    bTrackingMode : BOOL := FALSE; // 0 ACU转自跟踪；1 自己转
    bSearchType : BOOL := FALSE; // 0 直线扫；1 螺旋扫
    rErrorThre : REAL := 3.0; // 扫描找到中心：√(Ua²+Ue²) 门限(V)，可视化可下发
    rStartThre : REAL := 0.5;
    rAzScanRange : REAL := 1.0;
    rElScanRange : REAL := 1.0;
    rStep : REAL := 0.0015;
    rEbN0LockThre : REAL := 20.0; // 扫描找到中心：Eb/N0 门限，可视化可下发
END_VAR
(* global variable list GVL_PhaseCal *)
{attribute 'qualified_only'}
VAR_GLOBAL
    (* Commands: non-retained. Never FORCE these or axis commands. *)
    xStart : BOOL;
    xAbort : BOOL;
    xReset : BOOL;
    (* Commissioning interlock: confirm aligned reads with the actual protocol first.
       recSize>=16 alone is NOT a frame/header/checksum verification. *)
    xRxAlignmentConfirmed : BOOL := FALSE;
    lrCurrentPhaseDeg : LREAL := 0;
    iPhaseDirection : INT := 0; (* unknown=0, CCW=+1, CW=-1 *)
    lrRadiusDeg : LREAL := 0.05; (* maximum radial distance, not each leg *)
    lrLegTimeSec : LREAL := 10;
    lrSettleSec : LREAL := 1;
    lrMinEbN0 : LREAL := 29;

    xReady, xBusy, xDone, xFault, xAborted : BOOL;
    xFitValid, xSuggestedValid : BOOL;
    uiError, uiFitError, uiState : UINT;
    udiSamples : UDINT;
    lrAzBias, lrElBias, lrRxAgeSec : LREAL;
    lrResponseAngleDeg, lrCorrectionDeg, lrSuggestedDeg : LREAL;
    lrCandidatePlusDeg, lrCandidateMinusDeg : LREAL;
    lrOrthErrorDeg, lrResidualAz, lrResidualEl : LREAL;
    lrKaa, lrKae, lrKea, lrKee : LREAL;

    (* SerialCom single writer; Canopen single reader. Even/odd sequence lock.
       Positions are PLC feedback at receive time, not sender timestamps. *)
    udiRxSeq : UDINT;
    uiReadSize, uiSerialError : UINT;
    udiReadCount, udiShortReadCount : UDINT;
    lrRxUa, lrRxUe, lrRxEbN0, lrRxAz, lrRxEl : LREAL;
    xRxLock : BOOL;
END_VAR
    TASK MainTask(INTERVAL := T#50ms, PRIORITY := 10);
    TASK SerialCom(INTERVAL := T#5ms, PRIORITY := 1);
    TASK Canopen(INTERVAL := T#10ms, PRIORITY := 0);
    TASK Task(INTERVAL := T#50ms, PRIORITY := 31);
    TASK VISU_TASK(INTERVAL := T#100ms, PRIORITY := 31);
    PROGRAM Modbus_Slave WITH MainTask : Modbus_Slave;
    PROGRAM READ_485 WITH SerialCom : READ_485;
    PROGRAM GPRMC_1 WITH SerialCom : GPRMC_1;
    PROGRAM TimeAdd WITH Canopen : TimeAdd;
    PROGRAM AutoTrackingCal WITH Canopen : AutoTrackingCal;
    PROGRAM El_ctrl_1 WITH Canopen : El_ctrl_1;
    PROGRAM Az_ctrl_1 WITH Canopen : Az_ctrl_1;
    PROGRAM Ti_ctrl_1 WITH Canopen : Ti_ctrl_1;
    PROGRAM RealTimePosCal WITH Canopen : RealTimePosCal;
    PROGRAM SecurityCheck WITH Canopen : SecurityCheck;
    PROGRAM VisuElems.Visu_Prg WITH VISU_TASK : VisuElems.Visu_Prg;
  END_RESOURCE
END_CONFIGURATION

CONFIGURATION GCAN_IoDrv
END_CONFIGURATION

CONFIGURATION GCAN_IoMDP
END_CONFIGURATION

CONFIGURATION GC5016_Digital_Input_Output
END_CONFIGURATION

CONFIGURATION CANbus
END_CONFIGURATION

CONFIGURATION CANopen_Manager
END_CONFIGURATION

CONFIGURATION eDriver_El
END_CONFIGURATION

CONFIGURATION eDriver_Az
END_CONFIGURATION

CONFIGURATION eDriver_Ti
END_CONFIGURATION

CONFIGURATION SoftMotion General Axis Pool
END_CONFIGURATION
